KUKA KRL program: MyProgram_187().src

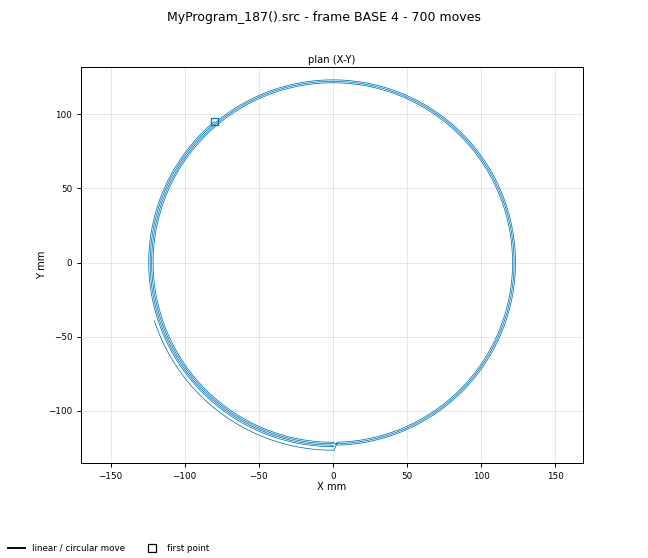
[picture p0: tool path of MyProgram_187().src in frame BASE 4, 700 of 700 moves have a stored position in this frame; points joined in program order, loops and branches not executed]
&ACCESS RVP
&REL 1
&PARAM TEMPLATE = C:\KRC\Roboter\Template\vorgabe
&PARAM EDITMASK = *
DEF MyProgram_187()
; ---- Setting reference (Base) ----
$BASE = BASE_DATA[4]

; --------------------------
; ---- Setting tool (TCP) ----
$TOOL = TOOL_DATA[3]
; --------------------------

$VEL.CP = VEL_APROX_PRINT
Startdeposition()
$VEL.CP = VEL_PRINT
LIN {X -79.8891,Y 95.1931,Z 136,A 126.8253,B 24.9437,C -1.7328,E1 24.8952,E2 319.3124} C_DIS
LIN {X -82.9171,Y 92.5676,Z 136,A 128.0656,B 24.9458,C -1.7009,E1 24.8928,E2 318.1432} C_DIS
LIN {X -85.2683,Y 90.4064,Z 136,A 130.1742,B 24.9442,C -1.7263,E1 24.8883,E2 315.9655} C_DIS
LIN {X -88.1797,Y 87.569,Z 136,A 131.451,B 24.9462,C -1.6946,E1 24.8859,E2 314.7588} C_DIS
LIN {X -91.7827,Y 83.7859,Z 136,A 133.7953,B 24.9468,C -1.6855,E1 24.8815,E2 312.4257} C_DIS
LIN {X -93.7322,Y 81.5983,Z 136,A 135.6415,B 24.9456,C -1.7044,E1 24.878,E2 310.5264} C_DIS
LIN {X -96.8546,Y 77.8667,Z 136,A 137.691,B 24.9465,C -1.6896,E1 24.8744,E2 308.5025} C_DIS
LIN {X -99.4155,Y 74.57,Z 136,A 139.5341,B 24.9471,C -1.6807,E1 24.8713,E2 306.6719} C_DIS
LIN {X -101.7751,Y 71.316,Z 136,A 141.5268,B 24.947,C -1.6818,E1 24.868,E2 304.6668} C_DIS
LIN {X -106.6362,Y 63.8183,Z 136,A 145.6095,B 24.9478,C -1.6682,E1 24.862,E2 300.5958} C_DIS
LIN {X -108.656,Y 60.3149,Z 136,A 148.5211,B 24.9452,C -1.71,E1 24.8579,E2 297.5692} C_DIS
LIN {X -111.8576,Y 54.1463,Z 136,A 150.5626,B 24.9491,C -1.6478,E1 24.8555,E2 295.6649} C_DIS
LIN {X -113.7433,Y 50.0655,Z 136,A 152.8918,B 24.9488,C -1.6529,E1 24.8528,E2 293.3109} C_DIS
LIN {X -115.0922,Y 46.8781,Z 136,A 154.451,B 24.9492,C -1.6463,E1 24.8511,E2 291.7587} C_DIS
LIN {X -116.506,Y 43.2441,Z 136,A 156.1505,B 24.9498,C -1.6363,E1 24.8494,E2 290.0735} C_DIS
LIN {X -117.7616,Y 39.6986,Z 136,A 157.9661,B 24.9499,C -1.6345,E1 24.8478,E2 288.252} C_DIS
LIN {X -119.6271,Y 33.6598,Z 136,A 160.8557,B 24.9506,C -1.624,E1 24.8455,E2 285.3706} C_DIS
LIN {X -120.6131,Y 29.9417,Z 136,A 162.772,B 24.9506,C -1.6246,E1 24.8441,E2 283.4416} C_DIS
LIN {X -122.2013,Y 22.6033,Z 136,A 166.0422,B 24.9517,C -1.6048,E1 24.8423,E2 280.1995} C_DIS
LIN {X -122.7677,Y 19.2815,Z 136,A 168.2135,B 24.9504,C -1.6274,E1 24.8413,E2 277.9615} C_DIS
LIN {X -123.363,Y 15.0101,Z 136,A 169.4402,B 24.9528,C -1.5868,E1 24.8409,E2 276.8241} C_DIS
LIN {X -123.9667,Y 8.7196,Z 136,A 172.4895,B 24.953,C -1.5832,E1 24.8402,E2 273.7651} C_DIS
LIN {X -124.135,Y 5.8576,Z 136,A 174.6101,B 24.9512,C -1.6146,E1 24.8399,E2 271.5569} C_DIS
LIN {X -124.2692,Y 0.9531,Z 136,A 176.6101,B 24.9523,C -1.5954,E1 24.8398,E2 269.5907} C_DIS
LIN {X -124.2442,Y -2.7393,Z 136,A 177.8627,B 24.9538,C -1.5697,E1 24.8398,E2 268.3918} C_DIS
LIN {X -124.1486,Y -5.5878,Z 136,A 179.9613,B 24.952,C -1.6006,E1 24.8402,E2 266.2069} C_DIS
LIN {X -123.821,Y -10.5841,Z 136,A -178.8273,B 24.9553,C -1.544,E1 24.8404,E2 265.1232} C_DIS
LIN {X -123.4086,Y -14.6276,Z 136,A -176.2872,B 24.954,C -1.5675,E1 24.8412,E2 262.5116} C_DIS
LIN {X -122.8522,Y -18.7364,Z 136,A -174.2614,B 24.954,C -1.5665,E1 24.842,E2 260.4763} C_DIS
LIN {X -122.3029,Y -22.0373,Z 136,A -172.7355,B 24.9544,C -1.5608,E1 24.8427,E2 258.9548} C_DIS
LIN {X -121.6747,Y -25.2814,Z 136,A -171.4403,B 24.9552,C -1.5458,E1 24.8434,E2 257.6879} C_DIS
LIN {X -120.8012,Y -29.1664,Z 136,A -169.6992,B 24.9558,C -1.5357,E1 24.8445,E2 255.9605} C_DIS
LIN {X -120.0039,Y -32.2916,Z 136,A -168.1059,B 24.9558,C -1.5359,E1 24.8457,E2 254.3576} C_DIS
LIN {X -118.874,Y -36.2296,Z 136,A -166.2328,B 24.9562,C -1.5293,E1 24.8472,E2 252.4893} C_DIS
LIN {X -117.8387,Y -39.4671,Z 136,A -164.6808,B 24.9565,C -1.5239,E1 24.8485,E2 250.9413} C_DIS
LIN {X -115.5921,Y -45.634,Z 136,A -161.576,B 24.9568,C -1.5183,E1 24.8516,E2 247.8323} C_DIS
LIN {X -114.1378,Y -49.1543,Z 136,A -159.2051,B 24.9555,C -1.5411,E1 24.8542,E2 245.3941} C_DIS
LIN {X -112.087,Y -53.6662,Z 136,A -157.5832,B 24.9576,C -1.5044,E1 24.8561,E2 243.8508} C_DIS
LIN {X -110.4867,Y -56.8906,Z 136,A -155.7892,B 24.9576,C -1.5058,E1 24.8584,E2 242.0439} C_DIS
LIN {X -107.6039,Y -62.1724,Z 136,A -153.0618,B 24.9581,C -1.496,E1 24.8621,E2 239.3255} C_DIS
LIN {X -105.3899,Y -65.8561,Z 136,A -150.667,B 24.9573,C -1.5095,E1 24.8656,E2 236.8863} C_DIS
LIN {X -103.2575,Y -69.1515,Z 136,A -149.3057,B 24.9587,C -1.4843,E1 24.8677,E2 235.5781} C_DIS
LIN {X -101.0566,Y -72.3296,Z 136,A -147.4329,B 24.9587,C -1.4839,E1 24.8707,E2 233.6972} C_DIS
LIN {X -97.1018,Y -77.5583,Z 136,A -144.667,B 24.9598,C -1.4647,E1 24.8753,E2 230.9637} C_DIS
LIN {X -95.265,Y -79.8034,Z 136,A -142.5722,B 24.9581,C -1.4963,E1 24.8792,E2 228.7842} C_DIS
LIN {X -92.3581,Y -83.151,Z 136,A -141.2515,B 24.9602,C -1.4582,E1 24.8815,E2 227.548} C_DIS
LIN {X -90.2674,Y -85.4156,Z 136,A -139.6102,B 24.9598,C -1.4652,E1 24.8847,E2 225.883} C_DIS
LIN {X -87.4192,Y -88.3286,Z 136,A -137.2447,B 24.9588,C -1.4836,E1 24.8895,E2 223.4636} C_DIS
LIN {X -84.3632,Y -91.2522,Z 136,A -135.706,B 24.96,C -1.4605,E1 24.8925,E2 221.9737} C_DIS
LIN {X -81.1483,Y -94.122,Z 136,A -133.2473,B 24.959,C -1.4785,E1 24.8978,E2 219.4625} C_DIS
LIN {X -77.7238,Y -96.9698,Z 136,A -131.922,B 24.9611,C -1.4407,E1 24.9005,E2 218.222} C_DIS
LIN {X -75.1964,Y -98.9426,Z 136,A -130.1587,B 24.9605,C -1.4513,E1 24.9045,E2 216.4273} C_DIS
LIN {X -71.5559,Y -101.6059,Z 136,A -128.1016,B 24.9608,C -1.4466,E1 24.9091,E2 214.374} C_DIS
LIN {X -68.0094,Y -104.0138,Z 136,A -126.0821,B 24.9608,C -1.4454,E1 24.9138,E2 212.3507} C_DIS
LIN {X -64.3396,Y -106.3222,Z 136,A -123.9135,B 24.9606,C -1.4504,E1 24.919,E2 210.1637} C_DIS
LIN {X -61.0887,Y -108.223,Z 136,A -122.3702,B 24.9612,C -1.4388,E1 24.9227,E2 208.6433} C_DIS
LIN {X -57.4568,Y -110.1925,Z 136,A -120.5659,B 24.9616,C -1.4315,E1 24.9271,E2 206.8512} C_DIS
LIN {X -54.7157,Y -111.5787,Z 136,A -119.0959,B 24.9616,C -1.4323,E1 24.9308,E2 205.3755} C_DIS
LIN {X -50.9574,Y -113.3444,Z 136,A -117.1344,B 24.9616,C -1.4323,E1 24.9358,E2 203.4092} C_DIS
LIN {X -47.7662,Y -114.7256,Z 136,A -115.5672,B 24.9618,C -1.4289,E1 24.9398,E2 201.8465} C_DIS
LIN {X -44.3758,Y -116.0812,Z 136,A -113.7716,B 24.9616,C -1.4325,E1 24.9445,E2 200.0384} C_DIS
LIN {X -40.7055,Y -117.4165,Z 136,A -112.0488,B 24.9618,C -1.4273,E1 24.9491,E2 198.3247} C_DIS
LIN {X -35.3019,Y -119.1534,Z 136,A -109.6672,B 24.9625,C -1.414,E1 24.9553,E2 195.9703} C_DIS
LIN {X -28.6712,Y -120.9205,Z 136,A -106.2014,B 24.9619,C -1.4265,E1 24.9648,E2 192.4698} C_DIS
LIN {X -24.5204,Y -121.8295,Z 136,A -104.3549,B 24.9622,C -1.4202,E1 24.9698,E2 190.636} C_DIS
LIN {X -20.6183,Y -122.5501,Z 136,A -102.4802,B 24.9622,C -1.4218,E1 24.975,E2 188.7557} C_DIS
LIN {X -16.3953,Y -123.1864,Z 136,A -100.6001,B 24.9624,C -1.417,E1 24.9801,E2 186.8853} C_DIS
LIN {X -13.0699,Y -123.5835,Z 136,A -98.9872,B 24.9622,C -1.4201,E1 24.9846,E2 185.2641} C_DIS
LIN {X -9.0853,Y -123.94,Z 136,A -97.1631,B 24.9622,C -1.4191,E1 24.9897,E2 183.4417} C_DIS
LIN {X -5.3221,Y -124.1595,Z 136,A -95.3481,B 24.9621,C -1.4229,E1 24.9948,E2 181.617} C_DIS
LIN {X -1.8056,Y -124.2598,Z 136,A -93.7695,B 24.9621,C -1.4211,E1 24.9992,E2 180.0426} C_DIS
LIN {X 0.8741,Y -124.2669,Z 136,A -92.7926,B 24.9628,C -1.4088,E1 25.0018,E2 179.0948} C_DIS
Enddeposition()
LIN {X 0.8741,Y -124.2669,Z 136,A -92.7926,B 24.9628,C -1.4088,E1 25.0018,E2 179.0948} C_DIS
Startdeposition()
$VEL.CP = VEL_PRINT
LIN {X -0.7971,Y -123.2805,Z 136,A -94.1303,B 24.9633,C -1.399,E1 24.998,E2 180.4558} C_DIS
LIN {X -4.8298,Y -123.1883,Z 136,A -95.9638,B 24.9633,C -1.4007,E1 24.9929,E2 182.2855} C_DIS
LIN {X -8.7858,Y -122.9696,Z 136,A -97.8638,B 24.9633,C -1.3979,E1 24.9876,E2 184.1928} C_DIS
LIN {X -13.0721,Y -122.5879,Z 136,A -99.8139,B 24.9633,C -1.4004,E1 24.9822,E2 186.1379} C_DIS
LIN {X -17.0591,Y -122.0974,Z 136,A -101.7751,B 24.9635,C -1.3964,E1 24.9767,E2 188.1103} C_DIS
LIN {X -20.0684,Y -121.6386,Z 136,A -103.1354,B 24.9633,C -1.3993,E1 24.973,E2 189.4648} C_DIS
LIN {X -23.7259,Y -120.9796,Z 136,A -104.9841,B 24.9636,C -1.3943,E1 24.9679,E2 191.3275} C_DIS
LIN {X -27.3955,Y -120.2003,Z 136,A -106.8949,B 24.9639,C -1.3874,E1 24.9626,E2 193.2571} C_DIS
LIN {X -30.6506,Y -119.4122,Z 136,A -108.2094,B 24.9633,C -1.3995,E1 24.9592,E2 194.5446} C_DIS
LIN {X -38.1177,Y -117.2435,Z 136,A -111.681,B 24.9628,C -1.4087,E1 24.9499,E2 198.0003} C_DIS
LIN {X -41.2854,Y -116.1655,Z 136,A -113.3984,B 24.9632,C -1.4025,E1 24.9453,E2 199.7358} C_DIS
LIN {X -44.7539,Y -114.8724,Z 136,A -115.0596,B 24.9629,C -1.4069,E1 24.941,E2 201.39} C_DIS
LIN {X -48.0441,Y -113.5371,Z 136,A -116.5953,B 24.9626,C -1.4139,E1 24.9371,E2 202.9126} C_DIS
LIN {X -50.4756,Y -112.4758,Z 136,A -117.9131,B 24.9626,C -1.4114,E1 24.9337,E2 204.2395} C_DIS
LIN {X -53.3978,Y -111.1185,Z 136,A -119.3608,B 24.9625,C -1.4154,E1 24.9301,E2 205.6812} C_DIS
LIN {X -56.2779,Y -109.6882,Z 136,A -120.8925,B 24.9625,C -1.4156,E1 24.9262,E2 207.2165} C_DIS
LIN {X -59.2874,Y -108.0931,Z 136,A -122.5495,B 24.9625,C -1.4144,E1 24.9221,E2 208.8812} C_DIS
LIN {X -62.877,Y -106.0443,Z 136,A -124.6374,B 24.9628,C -1.4095,E1 24.9171,E2 210.9869} C_DIS
LIN {X -66.1805,Y -104.0157,Z 136,A -126.3077,B 24.9623,C -1.4183,E1 24.9131,E2 212.6416} C_DIS
LIN {X -69.6137,Y -101.7496,Z 136,A -128.2574,B 24.9623,C -1.4197,E1 24.9086,E2 214.5944} C_DIS
LIN {X -73.3032,Y -99.1252,Z 136,A -130.3531,B 24.962,C -1.4237,E1 24.9039,E2 216.6879} C_DIS
LIN {X -76.6207,Y -96.5833,Z 136,A -132.9382,B 24.9634,C -1.3985,E1 24.8981,E2 219.3426} C_DIS
LIN {X -80.6051,Y -93.2838,Z 136,A -134.6338,B 24.9614,C -1.4349,E1 24.8946,E2 220.9581} C_DIS
LIN {X -83.5872,Y -90.6214,Z 136,A -137.0973,B 24.9627,C -1.4116,E1 24.8894,E2 223.487} C_DIS
LIN {X -86.899,Y -87.4504,Z 136,A -138.5028,B 24.9607,C -1.4486,E1 24.8868,E2 224.8104} C_DIS
LIN {X -89.289,Y -85.0091,Z 136,A -140.3163,B 24.9611,C -1.4419,E1 24.8832,E2 226.6476} C_DIS
LIN {X -94.242,Y -79.483,Z 136,A -143.5737,B 24.9602,C -1.4584,E1 24.8772,E2 229.8803} C_DIS
LIN {X -98.2148,Y -74.5182,Z 136,A -146.4389,B 24.9595,C -1.4696,E1 24.8723,E2 232.7324} C_DIS
LIN {X -99.7531,Y -72.4455,Z 136,A -147.9432,B 24.9601,C -1.459,E1 24.8697,E2 234.2692} C_DIS
LIN {X -102.2995,Y -68.8039,Z 136,A -150.822,B 24.9618,C -1.4286,E1 24.8651,E2 237.2347} C_DIS
LIN {X -105.4462,Y -63.8758,Z 136,A -153.3873,B 24.961,C -1.4425,E1 24.8614,E2 239.78} C_DIS
LIN {X -107.9909,Y -59.4732,Z 136,A -154.8402,B 24.9585,C -1.489,E1 24.8596,E2 241.1298} C_DIS
LIN {X -109.8808,Y -55.8996,Z 136,A -156.9074,B 24.9586,C -1.486,E1 24.8569,E2 243.2152} C_DIS
LIN {X -111.277,Y -53.0659,Z 136,A -159.3366,B 24.9607,C -1.4482,E1 24.8539,E2 245.7475} C_DIS
LIN {X -113.7429,Y -47.5514,Z 136,A -161.0675,B 24.9577,C -1.5034,E1 24.8521,E2 247.3566} C_DIS
LIN {X -116.1405,Y -41.3547,Z 136,A -164.2218,B 24.9573,C -1.5096,E1 24.8489,E2 250.5139} C_DIS
LIN {X -116.9716,Y -38.9387,Z 136,A -165.5697,B 24.9575,C -1.5062,E1 24.8477,E2 251.8776} C_DIS
LIN {X -118.0764,Y -35.4541,Z 136,A -167.3797,B 24.9575,C -1.5065,E1 24.8462,E2 253.6972} C_DIS
LIN {X -119.1135,Y -31.7896,Z 136,A -169.0301,B 24.9569,C -1.5172,E1 24.845,E2 255.3316} C_DIS
LIN {X -120.0435,Y -28.082,Z 136,A -170.9327,B 24.9569,C -1.5172,E1 24.8437,E2 257.2453} C_DIS
LIN {X -121.5095,Y -20.842,Z 136,A -174.1659,B 24.9557,C -1.5369,E1 24.842,E2 260.4509} C_DIS
LIN {X -122.1588,Y -16.6207,Z 136,A -176.9281,B 24.9573,C -1.5096,E1 24.8409,E2 263.2947} C_DIS
LIN {X -122.6999,Y -11.9764,Z 136,A -178.1992,B 24.9547,C -1.5557,E1 24.8406,E2 264.4634} C_DIS
LIN {X -123.0439,Y -7.6728,Z 136,A 179.2812,B 24.9556,C -1.5399,E1 24.84,E2 267.0358} C_DIS
LIN {X -123.2096,Y -4.2848,Z 136,A 177.075,B 24.9568,C -1.5179,E1 24.8398,E2 269.3077} C_DIS
LIN {X -123.2763,Y 1.43,Z 136,A 175.325,B 24.9541,C -1.5656,E1 24.8398,E2 270.9546} C_DIS
LIN {X -123.1001,Y 6.7344,Z 136,A 172.8345,B 24.9537,C -1.5726,E1 24.8401,E2 273.4433} C_DIS
LIN {X -122.5522,Y 13.4038,Z 136,A 169.7573,B 24.953,C -1.5842,E1 24.8408,E2 276.5113} C_DIS
LIN {X -121.7875,Y 19.1446,Z 136,A 166.9893,B 24.9526,C -1.5897,E1 24.8419,E2 279.2827} C_DIS
LIN {X -121.2402,Y 22.3575,Z 136,A 164.5557,B 24.9547,C -1.5551,E1 24.8432,E2 281.8134} C_DIS
LIN {X -120.0973,Y 27.8462,Z 136,A 162.8245,B 24.952,C -1.6011,E1 24.8442,E2 283.445} C_DIS
LIN {X -119.3463,Y 30.9102,Z 136,A 161.235,B 24.952,C -1.6005,E1 24.8452,E2 285.0453} C_DIS
LIN {X -118.0768,Y 35.447,Z 136,A 158.561,B 24.9528,C -1.5866,E1 24.8474,E2 287.7678} C_DIS
LIN {X -116.784,Y 39.5023,Z 136,A 157.1951,B 24.9509,C -1.6193,E1 24.8485,E2 289.0635} C_DIS
LIN {X -115.2983,Y 43.6472,Z 136,A 155.0459,B 24.9507,C -1.6213,E1 24.8506,E2 291.2201} C_DIS
LIN {X -113.8043,Y 47.4042,Z 136,A 153.1553,B 24.9504,C -1.6267,E1 24.8526,E2 293.1085} C_DIS
LIN {X -112.4721,Y 50.4839,Z 136,A 151.5761,B 24.9502,C -1.6306,E1 24.8543,E2 294.687} C_DIS
LIN {X -111.1031,Y 53.43,Z 136,A 149.5201,B 24.9513,C -1.6115,E1 24.8569,E2 296.7995} C_DIS
LIN {X -109.2176,Y 57.1847,Z 136,A 147.6227,B 24.9508,C -1.6198,E1 24.8593,E2 298.6874} C_DIS
LIN {X -107.2843,Y 60.7392,Z 136,A 146.388,B 24.9488,C -1.6534,E1 24.8609,E2 299.8486} C_DIS
LIN {X -102.6336,Y 68.3036,Z 136,A 142.0902,B 24.9485,C -1.6578,E1 24.8673,E2 304.1578} C_DIS
LIN {X -100.536,Y 71.3559,Z 136,A 140.2133,B 24.9486,C -1.6558,E1 24.8703,E2 306.0487} C_DIS
LIN {X -97.7397,Y 75.1402,Z 136,A 138.1224,B 24.948,C -1.666,E1 24.8737,E2 308.1254} C_DIS
LIN {X -95.4028,Y 78.0854,Z 136,A 136.0344,B 24.9486,C -1.6558,E1 24.8775,E2 310.2475} C_DIS
LIN {X -93.3376,Y 80.5426,Z 136,A 135.0727,B 24.9469,C -1.6829,E1 24.8791,E2 311.1489} C_DIS
LIN {X -91.5279,Y 82.594,Z 136,A 133.137,B 24.9485,C -1.657,E1 24.8828,E2 313.1549} C_DIS
LIN {X -88.9686,Y 85.3443,Z 136,A 131.8356,B 24.9471,C -1.6809,E1 24.8853,E2 314.4052} C_DIS
LIN {X -85.0552,Y 89.2449,Z 136,A 129.4074,B 24.9463,C -1.6933,E1 24.89,E2 316.8139} C_DIS
LIN {X -82.7792,Y 91.3598,Z 136,A 127.5149,B 24.9473,C -1.6769,E1 24.894,E2 318.7531} C_DIS
LIN {X -80.0922,Y 93.7249,Z 136,A 126.0172,B 24.9466,C -1.688,E1 24.8972,E2 320.2302} C_DIS
LIN {X -75.2732,Y 97.6374,Z 136,A 123.1518,B 24.9461,C -1.6952,E1 24.9034,E2 323.0892} C_DIS
LIN {X -71.9619,Y 100.1029,Z 136,A 120.9433,B 24.9467,C -1.6864,E1 24.9084,E2 325.3265} C_DIS
LIN {X -69.2441,Y 102.0014,Z 136,A 119.1971,B 24.9471,C -1.6804,E1 24.9125,E2 327.0927} C_DIS
LIN {X -65.6679,Y 104.3395,Z 136,A 117.7502,B 24.9453,C -1.7081,E1 24.9158,E2 328.4783} C_DIS
LIN {X -62.2817,Y 106.3957,Z 136,A 115.7431,B 24.9456,C -1.7041,E1 24.9206,E2 330.501} C_DIS
LIN {X -58.7148,Y 108.4053,Z 136,A 113.8957,B 24.9452,C -1.7099,E1 24.9251,E2 332.34} C_DIS
LIN {X -55.6171,Y 110.0246,Z 136,A 112.3365,B 24.9448,C -1.7156,E1 24.929,E2 333.8899} C_DIS
LIN {X -51.8752,Y 111.8372,Z 136,A 110.3993,B 24.9447,C -1.7185,E1 24.9339,E2 335.8252} C_DIS
LIN {X -46.0929,Y 114.3417,Z 136,A 107.836,B 24.9433,C -1.7393,E1 24.9404,E2 338.3451} C_DIS
LIN {X -42.9145,Y 115.5727,Z 136,A 105.8955,B 24.9442,C -1.7252,E1 24.9455,E2 340.323} C_DIS
LIN {X -38.5445,Y 117.1029,Z 136,A 103.7789,B 24.9439,C -1.7295,E1 24.9511,E2 342.4335} C_DIS
LIN {X -35.6805,Y 118.0071,Z 136,A 102.3388,B 24.9439,C -1.7291,E1 24.9549,E2 343.8771} C_DIS
LIN {X -29.2711,Y 119.758,Z 136,A 99.4324,B 24.9432,C -1.7406,E1 24.9627,E2 346.7607} C_DIS
LIN {X -27.0063,Y 120.2889,Z 136,A 97.6434,B 24.9452,C -1.7093,E1 24.9678,E2 348.6262} C_DIS
LIN {X -22.9703,Y 121.124,Z 136,A 96.5296,B 24.9428,C -1.7475,E1 24.9706,E2 349.6506} C_DIS
LIN {X -20.395,Y 121.5841,Z 136,A 94.3114,B 24.9457,C -1.7026,E1 24.977,E2 351.9775} C_DIS
LIN {X -15.2822,Y 122.3339,Z 136,A 92.6842,B 24.9433,C -1.7394,E1 24.9813,E2 353.5186} C_DIS
LIN {X -10.9994,Y 122.7928,Z 136,A 90.4986,B 24.9438,C -1.732,E1 24.9874,E2 355.723} C_DIS
LIN {X -7.0479,Y 123.0824,Z 136,A 88.6722,B 24.9437,C -1.7334,E1 24.9925,E2 357.5466} C_DIS
LIN {X -3.1815,Y 123.2421,Z 136,A 86.9936,B 24.9433,C -1.7395,E1 24.9971,E2 359.2109} C_DIS
LIN {X 0.5109,Y 123.2821,Z 136,A 85.2323,B 24.9434,C -1.7378,E1 25.002,E2 360.9764} C_DIS
LIN {X 4.5588,Y 123.1989,Z 136,A 83.3503,B 24.9434,C -1.738,E1 25.0073,E2 362.8575} C_DIS
LIN {X 8.0968,Y 123.0178,Z 136,A 81.6549,B 24.9435,C -1.7357,E1 25.012,E2 364.5577} C_DIS
LIN {X 11.8511,Y 122.7119,Z 136,A 79.9012,B 24.9435,C -1.7354,E1 25.0169,E2 366.3111} C_DIS
LIN {X 16.386,Y 122.1895,Z 136,A 77.8547,B 24.9434,C -1.7385,E1 25.0225,E2 368.3487} C_DIS
LIN {X 20.1788,Y 121.6202,Z 136,A 75.7807,B 24.9443,C -1.7242,E1 25.0284,E2 370.4544} C_DIS
LIN {X 23.9354,Y 120.9387,Z 136,A 74.2502,B 24.9436,C -1.7349,E1 25.0325,E2 371.9578} C_DIS
LIN {X 26.8973,Y 120.3141,Z 136,A 73.0086,B 24.9431,C -1.742,E1 25.0358,E2 373.181} C_DIS
LIN {X 29.837,Y 119.6187,Z 136,A 70.7055,B 24.9459,C -1.6988,E1 25.0423,E2 375.5829} C_DIS
LIN {X 35.0837,Y 118.1861,Z 136,A 69.1007,B 24.9432,C -1.7406,E1 25.0464,E2 377.0863} C_DIS
LIN {X 37.5544,Y 117.4234,Z 136,A 67.7868,B 24.9436,C -1.7343,E1 25.0499,E2 378.4126} C_DIS
LIN {X 41.1043,Y 116.2308,Z 136,A 65.8924,B 24.9442,C -1.7254,E1 25.0549,E2 380.3243} C_DIS
LIN {X 44.6198,Y 114.9246,Z 136,A 64.3147,B 24.9438,C -1.7316,E1 25.059,E2 381.884} C_DIS
LIN {X 47.8018,Y 113.6383,Z 136,A 62.7298,B 24.9438,C -1.7304,E1 25.0631,E2 383.468} C_DIS
LIN {X 51.0017,Y 112.2405,Z 136,A 60.8741,B 24.9447,C -1.7173,E1 25.0679,E2 385.3501} C_DIS
LIN {X 54.6188,Y 110.5231,Z 136,A 59.218,B 24.9442,C -1.7248,E1 25.072,E2 386.984} C_DIS
LIN {X 57.6727,Y 108.9613,Z 136,A 57.6108,B 24.9444,C -1.7221,E1 25.076,E2 388.5933} C_DIS
LIN {X 61.2582,Y 106.9883,Z 136,A 55.5187,B 24.9452,C -1.7101,E1 25.0811,E2 390.7074} C_DIS
LIN {X 64.532,Y 105.0459,Z 136,A 53.9147,B 24.9449,C -1.7154,E1 25.0849,E2 392.2939} C_DIS
LIN {X 67.9392,Y 102.8752,Z 136,A 52.0488,B 24.945,C -1.7129,E1 25.0893,E2 394.1596} C_DIS
LIN {X 71.3905,Y 100.5114,Z 136,A 50.0353,B 24.9454,C -1.7062,E1 25.0939,E2 396.1819} C_DIS
LIN {X 75.2954,Y 97.6192,Z 136,A 47.5381,B 24.9464,C -1.6906,E1 25.0995,E2 398.7071} C_DIS
LIN {X 78.0673,Y 95.4176,Z 136,A 46.4356,B 24.945,C -1.7139,E1 25.1018,E2 399.7504} C_DIS
LIN {X 80.3223,Y 93.5274,Z 136,A 44.8089,B 24.9459,C -1.6985,E1 25.1053,E2 401.4072} C_DIS
LIN {X 83.5894,Y 90.6194,Z 136,A 42.8267,B 24.946,C -1.6968,E1 25.1094,E2 403.3854} C_DIS
LIN {X 86.6269,Y 87.7208,Z 136,A 40.8362,B 24.9464,C -1.6907,E1 25.1134,E2 405.382} C_DIS
LIN {X 89.9028,Y 84.3589,Z 136,A 38.4815,B 24.9473,C -1.6773,E1 25.118,E2 407.7581} C_DIS
LIN {X 92.5137,Y 81.4879,Z 136,A 36.8883,B 24.9469,C -1.6835,E1 25.1209,E2 409.3296} C_DIS
LIN {X 95.2199,Y 78.309,Z 136,A 34.9921,B 24.947,C -1.681,E1 25.1243,E2 411.223} C_DIS
LIN {X 97.7627,Y 75.1102,Z 136,A 33.0687,B 24.9474,C -1.6751,E1 25.1276,E2 413.1511} C_DIS
LIN {X 100.2457,Y 71.7622,Z 136,A 31.1524,B 24.9477,C -1.6713,E1 25.1308,E2 415.0673} C_DIS
LIN {X 102.7626,Y 68.1103,Z 136,A 29.0612,B 24.9481,C -1.6644,E1 25.1341,E2 417.1643} C_DIS
LIN {X 105.1582,Y 64.349,Z 136,A 27.0529,B 24.9482,C -1.6621,E1 25.137,E2 419.168} C_DIS
LIN {X 107.309,Y 60.6951,Z 136,A 25.0597,B 24.9486,C -1.6555,E1 25.1398,E2 421.1663} C_DIS
LIN {X 109.3355,Y 56.9601,Z 136,A 23.2234,B 24.9486,C -1.657,E1 25.1422,E2 422.9896} C_DIS
LIN {X 110.9331,Y 53.7859,Z 136,A 21.0139,B 24.9506,C -1.6244,E1 25.145,E2 425.264} C_DIS
LIN {X 112.7251,Y 49.9181,Z 136,A 19.6538,B 24.949,C -1.6496,E1 25.1465,E2 426.5573} C_DIS
LIN {X 113.8281,Y 47.3473,Z 136,A 18.286,B 24.9495,C -1.6424,E1 25.148,E2 427.9345} C_DIS
LIN {X 115.3108,Y 43.6138,Z 136,A 16.4069,B 24.9498,C -1.6362,E1 25.1499,E2 429.8178} C_DIS
LIN {X 116.4617,Y 40.4383,Z 136,A 14.9034,B 24.9499,C -1.6348,E1 25.1513,E2 431.3161} C_DIS
LIN {X 118.8182,Y 32.8778,Z 136,A 11.1306,B 24.9509,C -1.6188,E1 25.1544,E2 435.1052} C_DIS
LIN {X 120.2244,Y 27.2899,Z 136,A 8.4179,B 24.9515,C -1.6086,E1 25.1562,E2 437.8262} C_DIS
LIN {X 121.6217,Y 20.1694,Z 136,A 5.2082,B 24.9517,C -1.6061,E1 25.1578,E2 441.0232} C_DIS
LIN {X 122.2843,Y 15.6626,Z 136,A 3.2015,B 24.9517,C -1.6048,E1 25.1586,E2 443.021} C_DIS
LIN {X 122.5732,Y 13.209,Z 136,A 1.9814,B 24.9522,C -1.5975,E1 25.159,E2 444.2512} C_DIS
LIN {X 122.9105,Y 9.5956,Z 136,A 0.1999,B 24.9528,C -1.5872,E1 25.1594,E2 446.0464} C_DIS
LIN {X 123.1431,Y 5.8773,Z 136,A -1.4797,B 24.953,C -1.5842,E1 25.1597,E2 447.7231} C_DIS
LIN {X 123.268,Y 1.9235,Z 136,A -3.2531,B 24.9531,C -1.5814,E1 25.1597,E2 449.4925} C_DIS
LIN {X 123.2658,Y -2.0555,Z 136,A -5.0751,B 24.9534,C -1.5767,E1 25.1597,E2 451.3146} C_DIS
LIN {X 123.1436,Y -5.8679,Z 136,A -6.9014,B 24.9539,C -1.5682,E1 25.1595,E2 453.1502} C_DIS
LIN {X 122.8768,Y -10.0051,Z 136,A -8.8377,B 24.9543,C -1.5614,E1 25.1592,E2 455.0911} C_DIS
LIN {X 122.4882,Y -13.9882,Z 136,A -10.6975,B 24.9547,C -1.5552,E1 25.1586,E2 456.9544} C_DIS
LIN {X 122.002,Y -17.7267,Z 136,A -12.4439,B 24.955,C -1.5498,E1 25.1579,E2 458.7034} C_DIS
LIN {X 121.3479,Y -21.7557,Z 136,A -14.2306,B 24.955,C -1.5492,E1 25.1571,E2 460.481} C_DIS
LIN {X 120.4026,Y -26.4967,Z 136,A -16.5301,B 24.9556,C -1.5391,E1 25.1558,E2 462.7907} C_DIS
LIN {X 119.5011,Y -30.3002,Z 136,A -18.267,B 24.9557,C -1.5373,E1 25.1546,E2 464.5219} C_DIS
LIN {X 118.5106,Y -33.9753,Z 136,A -20.9295,B 24.9586,C -1.4867,E1 25.1525,E2 467.2885} C_DIS
LIN {X 116.6947,Y -39.7662,Z 136,A -22.7395,B 24.9562,C -1.5284,E1 25.151,E2 468.9899} C_DIS
LIN {X 115.365,Y -43.4691,Z 136,A -24.6424,B 24.9568,C -1.5189,E1 25.1492,E2 470.9045} C_DIS
LIN {X 112.7492,Y -49.8642,Z 136,A -27.6899,B 24.9568,C -1.5171,E1 25.146,E2 473.9394} C_DIS
LIN {X 111.2087,Y -53.209,Z 136,A -29.4819,B 24.9574,C -1.5078,E1 25.1438,E2 475.7437} C_DIS
LIN {X 108.7471,Y -58.0782,Z 136,A -32.0419,B 24.9579,C -1.4989,E1 25.1406,E2 478.3112} C_DIS
LIN {X 107.4753,Y -60.3992,Z 136,A -33.3556,B 24.9584,C -1.491,E1 25.1387,E2 479.6367} C_DIS
LIN {X 105.2688,Y -64.1687,Z 136,A -35.7157,B 24.9596,C -1.4684,E1 25.1353,E2 482.0378} C_DIS
LIN {X 103.2715,Y -67.3356,Z 136,A -36.8724,B 24.9583,C -1.4927,E1 25.1336,E2 483.1314} C_DIS
LIN {X 100.3985,Y -71.5485,Z 136,A -39.3319,B 24.9589,C -1.4815,E1 25.1297,E2 485.6054} C_DIS
LIN {X 98.2955,Y -74.4107,Z 136,A -41.142,B 24.9596,C -1.4689,E1 25.1267,E2 487.4365} C_DIS
LIN {X 95.965,Y -77.3933,Z 136,A -43.0619,B 24.9603,C -1.4561,E1 25.1233,E2 489.3777} C_DIS
LIN {X 92.4118,Y -81.6032,Z 136,A -45.39,B 24.96,C -1.4609,E1 25.1191,E2 491.6838} C_DIS
LIN {X 89.487,Y -84.8007,Z 136,A -47.6304,B 24.9609,C -1.4445,E1 25.1147,E2 493.9532} C_DIS
LIN {X 87.2261,Y -87.1247,Z 136,A -49.0699,B 24.9609,C -1.4441,E1 25.1119,E2 495.3875} C_DIS
LIN {X 84.2892,Y -89.9694,Z 136,A -50.7809,B 24.9607,C -1.4489,E1 25.1085,E2 497.0801} C_DIS
LIN {X 80.1903,Y -93.6402,Z 136,A -53.4138,B 24.9612,C -1.4391,E1 25.1029,E2 499.7256} C_DIS
LIN {X 76.4504,Y -96.7186,Z 136,A -55.6152,B 24.9613,C -1.4366,E1 25.0982,E2 501.9248} C_DIS
LIN {X 72.9054,Y -99.4175,Z 136,A -58.3817,B 24.9634,C -1.3979,E1 25.0918,E2 504.7728} C_DIS
LIN {X 68.2172,Y -102.6913,Z 136,A -60.8335,B 24.9632,C -1.4026,E1 25.0861,E2 507.2054} C_DIS
LIN {X 64.1861,Y -105.2581,Z 136,A -62.1583,B 24.961,C -1.4424,E1 25.0832,E2 508.4318} C_DIS
LIN {X 60.242,Y -107.5637,Z 136,A -64.9452,B 24.963,C -1.4058,E1 25.0763,E2 511.2969} C_DIS
LIN {X 57.0538,Y -109.2863,Z 136,A -66.7555,B 24.9635,C -1.3968,E1 25.0717,E2 513.1234} C_DIS
LIN {X 53.1586,Y -111.2327,Z 136,A -68.1935,B 24.9621,C -1.4221,E1 25.0683,E2 514.4978} C_DIS
LIN {X 45.6218,Y -114.5316,Z 136,A -71.9656,B 24.9623,C -1.4188,E1 25.0586,E2 518.2687} C_DIS
LIN {X 43.1448,Y -115.4864,Z 136,A -73.2396,B 24.9625,C -1.4151,E1 25.0553,E2 519.5486} C_DIS
LIN {X 39.6073,Y -116.749,Z 136,A -76.0752,B 24.9653,C -1.3602,E1 25.0475,E2 522.5085} C_DIS
LIN {X 33.114,Y -118.7522,Z 136,A -78.0897,B 24.9627,C -1.4117,E1 25.0424,E2 524.3978} C_DIS
LIN {X 30.011,Y -119.5745,Z 136,A -80.1416,B 24.9642,C -1.3831,E1 25.0367,E2 526.5143} C_DIS
LIN {X 26.0247,Y -120.5045,Z 136,A -82.0179,B 24.9642,C -1.3826,E1 25.0315,E2 528.3893} C_DIS
LIN {X 22.0606,Y -121.2934,Z 136,A -83.2019,B 24.9625,C -1.4144,E1 25.0285,E2 529.4966} C_DIS
LIN {X 17.983,Y -121.9654,Z 136,A -85.3782,B 24.9633,C -1.4006,E1 25.0224,E2 531.7035} C_DIS
LIN {X 14.3981,Y -122.4393,Z 136,A -87.0795,B 24.9633,C -1.3986,E1 25.0177,E2 533.4083} C_DIS
LIN {X 10.4934,Y -122.8355,Z 136,A -88.8415,B 24.9633,C -1.4006,E1 25.0128,E2 535.1645} C_DIS
LIN {X 7.2186,Y -123.0719,Z 136,A -90.4395,B 24.9635,C -1.3965,E1 25.0083,E2 536.7715} C_DIS
LIN {X 3.2582,Y -123.24,Z 136,A -92.2671,B 24.9635,C -1.3965,E1 25.0032,E2 538.5986} C_DIS
LIN {X 3.2582,Y -123.24,Z 136,A -92.2671,B 24.9635,C -1.3965,E1 25.0032,E2 538.5986} C_DIS
Enddeposition()
LIN {X 0.8719,Y -122.2892,Z 136,A -93.284,B 24.9623,C -1.4181,E1 25.0005,E2 539.5643} C_DIS
Startdeposition()
$VEL.CP = VEL_PRINT
LIN {X 4.9775,Y -122.1922,Z 136,A -90.6693,B 24.9605,C -1.4516,E1 25.0081,E2 536.8707} C_DIS
LIN {X 8.8136,Y -121.9753,Z 136,A -88.8584,B 24.9605,C -1.4529,E1 25.0131,E2 535.0575} C_DIS
LIN {X 12.8168,Y -121.62,Z 136,A -86.953,B 24.9603,C -1.455,E1 25.0184,E2 533.1483} C_DIS
LIN {X 17.0537,Y -121.0985,Z 136,A -84.9998,B 24.9603,C -1.4541,E1 25.0238,E2 531.1989} C_DIS
LIN {X 20.7767,Y -120.5171,Z 136,A -83.3181,B 24.9605,C -1.4513,E1 25.0284,E2 529.5254} C_DIS
LIN {X 24.1435,Y -119.8864,Z 136,A -81.5449,B 24.96,C -1.4609,E1 25.0333,E2 527.7315} C_DIS
LIN {X 28.5926,Y -118.9036,Z 136,A -79.5211,B 24.9602,C -1.4576,E1 25.0388,E2 525.7185} C_DIS
LIN {X 32.0504,Y -118.0198,Z 136,A -77.7496,B 24.9598,C -1.4642,E1 25.0436,E2 523.9341} C_DIS
LIN {X 36.1049,Y -116.8423,Z 136,A -75.4997,B 24.959,C -1.4799,E1 25.0497,E2 521.6512} C_DIS
LIN {X 39.5336,Y -115.728,Z 136,A -74.131,B 24.9597,C -1.4662,E1 25.0533,E2 520.3173} C_DIS
LIN {X 42.9096,Y -114.5178,Z 136,A -72.5915,B 24.96,C -1.4616,E1 25.0573,E2 518.792} C_DIS
LIN {X 46.4141,Y -113.1452,Z 136,A -70.3755,B 24.9586,C -1.4864,E1 25.0631,E2 516.5223} C_DIS
LIN {X 49.5942,Y -111.7859,Z 136,A -69.1092,B 24.9594,C -1.4714,E1 25.0663,E2 515.2946} C_DIS
LIN {X 52.5031,Y -110.4492,Z 136,A -67.6604,B 24.9594,C -1.4714,E1 25.0699,E2 513.8497} C_DIS
LIN {X 55.296,Y -109.0776,Z 136,A -66.2834,B 24.9595,C -1.4698,E1 25.0733,E2 512.4801} C_DIS
LIN {X 60.3781,Y -106.351,Z 136,A -63.4126,B 24.9588,C -1.4829,E1 25.0804,E2 509.5867} C_DIS
LIN {X 63.9099,Y -104.2666,Z 136,A -61.374,B 24.9583,C -1.4924,E1 25.0853,E2 507.532} C_DIS
LIN {X 68.0469,Y -101.6151,Z 136,A -59.2113,B 24.9584,C -1.49,E1 25.0904,E2 505.3821} C_DIS
LIN {X 72.4362,Y -98.5342,Z 136,A -56.7343,B 24.9582,C -1.4935,E1 25.096,E2 502.9054} C_DIS
LIN {X 75.7369,Y -96.0207,Z 136,A -54.9435,B 24.9584,C -1.4901,E1 25.0999,E2 501.1292} C_DIS
LIN {X 78.3757,Y -93.8789,Z 136,A -52.6787,B 24.9563,C -1.5275,E1 25.1049,E2 498.7847} C_DIS
LIN {X 81.8848,Y -90.8351,Z 136,A -51.0323,B 24.9575,C -1.5059,E1 25.1083,E2 497.1959} C_DIS
LIN {X 84.884,Y -88.0384,Z 136,A -49.0987,B 24.9572,C -1.5112,E1 25.1122,E2 495.2578} C_DIS
LIN {X 88.0703,Y -84.851,Z 136,A -47.0279,B 24.957,C -1.5144,E1 25.1162,E2 493.1882} C_DIS
LIN {X 90.8819,Y -81.8325,Z 136,A -45.0659,B 24.9567,C -1.5209,E1 25.1199,E2 491.2197} C_DIS
LIN {X 93.522,Y -78.8016,Z 136,A -43.2143,B 24.9565,C -1.5243,E1 25.1233,E2 489.3685} C_DIS
LIN {X 95.8312,Y -75.9765,Z 136,A -41.1371,B 24.9551,C -1.5476,E1 25.127,E2 487.2461} C_DIS
LIN {X 98.2633,Y -72.8038,Z 136,A -39.701,B 24.9561,C -1.5306,E1 25.1293,E2 485.857} C_DIS
LIN {X 99.9625,Y -70.452,Z 136,A -38.2551,B 24.9556,C -1.5388,E1 25.1317,E2 484.3987} C_DIS
LIN {X 102.4791,Y -66.7387,Z 136,A -36.2252,B 24.9556,C -1.5412,E1 25.1348,E2 482.3734} C_DIS
LIN {X 104.9318,Y -62.812,Z 136,A -34.0658,B 24.9552,C -1.547,E1 25.1379,E2 480.2112} C_DIS
LIN {X 106.7464,Y -59.6764,Z 136,A -32.1027,B 24.9541,C -1.5656,E1 25.1407,E2 478.2144} C_DIS
LIN {X 108.3175,Y -56.7702,Z 136,A -30.9331,B 24.9549,C -1.551,E1 25.1421,E2 477.0854} C_DIS
LIN {X 109.9684,Y -53.5063,Z 136,A -29.2615,B 24.9548,C -1.554,E1 25.1442,E2 475.4156} C_DIS
LIN {X 111.4612,Y -50.3203,Z 136,A -27.5266,B 24.9542,C -1.5635,E1 25.1463,E2 473.6676} C_DIS
LIN {X 112.9516,Y -46.8781,Z 136,A -25.5663,B 24.9533,C -1.5793,E1 25.1484,E2 471.6809} C_DIS
LIN {X 114.8319,Y -42.0664,Z 136,A -23.3478,B 24.9534,C -1.5767,E1 25.1506,E2 469.481} C_DIS
LIN {X 116.0337,Y -38.6233,Z 136,A -21.4065,B 24.9524,C -1.594,E1 25.1523,E2 467.5098} C_DIS
LIN {X 117.0544,Y -35.4119,Z 136,A -20.0675,B 24.9528,C -1.5868,E1 25.1534,E2 466.1955} C_DIS
LIN {X 118.0661,Y -31.8768,Z 136,A -18.4651,B 24.9528,C -1.5862,E1 25.1546,E2 464.6035} C_DIS
LIN {X 118.8343,Y -28.88,Z 136,A -16.9694,B 24.9524,C -1.5933,E1 25.1556,E2 463.0999} C_DIS
LIN {X 119.7623,Y -24.7537,Z 136,A -15.257,B 24.9529,C -1.586,E1 25.1566,E2 461.4145} C_DIS
LIN {X 120.3764,Y -21.5671,Z 136,A -13.5391,B 24.952,C -1.601,E1 25.1575,E2 459.6713} C_DIS
LIN {X 120.8966,Y -18.431,Z 136,A -12.0712,B 24.9517,C -1.6048,E1 25.1581,E2 458.2031} C_DIS
LIN {X 121.4088,Y -14.6821,Z 136,A -10.2868,B 24.9514,C -1.6112,E1 25.1588,E2 456.4141} C_DIS
LIN {X 121.8134,Y -10.8367,Z 136,A -8.4373,B 24.9509,C -1.6191,E1 25.1593,E2 454.557} C_DIS
LIN {X 122.1019,Y -6.8698,Z 136,A -6.5522,B 24.9504,C -1.6263,E1 25.1596,E2 452.6661} C_DIS
LIN {X 122.2556,Y -3.0574,Z 136,A -4.8686,B 24.9504,C -1.6269,E1 25.1598,E2 450.9911} C_DIS
LIN {X 122.2941,Y 0.1575,Z 136,A -3.3587,B 24.9501,C -1.6321,E1 25.1598,E2 449.4781} C_DIS
LIN {X 122.2367,Y 3.7374,Z 136,A -1.6279,B 24.9496,C -1.6403,E1 25.1597,E2 447.7382} C_DIS
LIN {X 122.0481,Y 7.7441,Z 136,A 0.2394,B 24.9492,C -1.6458,E1 25.1594,E2 445.8689} C_DIS
LIN {X 121.7206,Y 11.8214,Z 136,A 2.0718,B 24.9492,C -1.6478,E1 25.1589,E2 444.0427} C_DIS
LIN {X 121.412,Y 14.6559,Z 136,A 3.807,B 24.9476,C -1.6725,E1 25.1583,E2 442.2597} C_DIS
LIN {X 120.9001,Y 18.4084,Z 136,A 4.9092,B 24.9494,C -1.644,E1 25.1579,E2 441.2311} C_DIS
LIN {X 120.5079,Y 20.83,Z 136,A 6.732,B 24.947,C -1.6818,E1 25.157,E2 439.3298} C_DIS
LIN {X 119.8092,Y 24.5228,Z 136,A 8.0435,B 24.9481,C -1.6646,E1 25.1563,E2 438.0666} C_DIS
LIN {X 118.6039,Y 29.8124,Z 136,A 10.5851,B 24.9476,C -1.6726,E1 25.1547,E2 435.5209} C_DIS
LIN {X 117.6952,Y 33.2192,Z 136,A 12.2077,B 24.9473,C -1.6762,E1 25.1535,E2 433.899} C_DIS
LIN {X 116.1078,Y 38.4006,Z 136,A 14.6875,B 24.947,C -1.681,E1 25.1514,E2 431.422} C_DIS
LIN {X 115.1035,Y 41.313,Z 136,A 16.1313,B 24.9468,C -1.6854,E1 25.1501,E2 429.976} C_DIS
LIN {X 113.9852,Y 44.3048,Z 136,A 17.6391,B 24.9464,C -1.6904,E1 25.1486,E2 428.4646} C_DIS
LIN {X 112.5172,Y 47.9153,Z 136,A 19.377,B 24.9464,C -1.6914,E1 25.1467,E2 426.7341} C_DIS
LIN {X 110.8369,Y 51.6805,Z 136,A 21.4794,B 24.9455,C -1.7056,E1 25.1442,E2 424.6096} C_DIS
LIN {X 109.0593,Y 55.3319,Z 136,A 23.2529,B 24.9455,C -1.7045,E1 25.1421,E2 422.8482} C_DIS
LIN {X 107.5335,Y 58.2465,Z 136,A 24.8419,B 24.9451,C -1.7112,E1 25.14,E2 421.2517} C_DIS
LIN {X 105.8235,Y 61.2975,Z 136,A 26.4818,B 24.9448,C -1.7157,E1 25.1377,E2 419.6096} C_DIS
LIN {X 103.6353,Y 64.9297,Z 136,A 28.5073,B 24.9444,C -1.723,E1 25.1347,E2 417.5772} C_DIS
LIN {X 101.3364,Y 68.4612,Z 136,A 30.4577,B 24.9441,C -1.727,E1 25.1317,E2 415.6271} C_DIS
LIN {X 98.8001,Y 72.074,Z 136,A 32.4961,B 24.9439,C -1.7308,E1 25.1284,E2 413.5897} C_DIS
LIN {X 96.3704,Y 75.2916,Z 136,A 34.4146,B 24.9435,C -1.7369,E1 25.1251,E2 411.6657} C_DIS
LIN {X 93.835,Y 78.4285,Z 136,A 36.2853,B 24.9432,C -1.7405,E1 25.1218,E2 409.7952} C_DIS
LIN {X 91.4307,Y 81.2185,Z 136,A 38.7915,B 24.9404,C -1.7835,E1 25.117,E2 407.1986} C_DIS
LIN {X 87.3589,Y 85.5828,Z 136,A 40.732,B 24.9428,C -1.747,E1 25.1134,E2 405.3527} C_DIS
LIN {X 84.3471,Y 88.5528,Z 136,A 42.6781,B 24.9426,C -1.7495,E1 25.1095,E2 403.4089} C_DIS
LIN {X 81.4078,Y 91.2623,Z 136,A 44.7061,B 24.9419,C -1.761,E1 25.1052,E2 401.3619} C_DIS
LIN {X 77.9399,Y 94.241,Z 136,A 47.6179,B 24.939,C -1.8033,E1 25.0988,E2 398.3612} C_DIS
LIN {X 72.9695,Y 98.14,Z 136,A 49.643,B 24.9418,C -1.7625,E1 25.0945,E2 396.44} C_DIS
LIN {X 69.8674,Y 100.372,Z 136,A 51.3738,B 24.9418,C -1.7627,E1 25.0906,E2 394.7147} C_DIS
LIN {X 66.9588,Y 102.3358,Z 136,A 53.1353,B 24.9412,C -1.7711,E1 25.0864,E2 392.9392} C_DIS
LIN {X 63.6274,Y 104.4398,Z 136,A 54.87,B 24.9414,C -1.7685,E1 25.0824,E2 391.2161} C_DIS
LIN {X 60.6134,Y 106.2168,Z 136,A 56.5145,B 24.9412,C -1.7712,E1 25.0784,E2 389.5702} C_DIS
LIN {X 57.58,Y 107.8919,Z 136,A 58.1065,B 24.9412,C -1.7719,E1 25.0745,E2 387.9811} C_DIS
LIN {X 54.4924,Y 109.482,Z 136,A 59.7777,B 24.9409,C -1.7762,E1 25.0703,E2 386.3043} C_DIS
LIN {X 51.2598,Y 111.0314,Z 136,A 61.4492,B 24.9408,C -1.7779,E1 25.0661,E2 384.6332} C_DIS
LIN {X 47.5551,Y 112.6688,Z 136,A 63.354,B 24.9406,C -1.7803,E1 25.0612,E2 382.7271} C_DIS
LIN {X 44.4683,Y 113.9217,Z 136,A 64.8665,B 24.9406,C -1.7796,E1 25.0573,E2 381.2197} C_DIS
LIN {X 41.2909,Y 115.1115,Z 136,A 66.4622,B 24.9406,C -1.7814,E1 25.0531,E2 379.6231} C_DIS
LIN {X 37.5223,Y 116.3948,Z 136,A 68.321,B 24.9404,C -1.7827,E1 25.0482,E2 377.7649} C_DIS
LIN {X 34.1434,Y 117.4302,Z 136,A 69.8554,B 24.9407,C -1.7781,E1 25.0441,E2 376.2439} C_DIS
LIN {X 30.0781,Y 118.5365,Z 136,A 71.9569,B 24.9402,C -1.7855,E1 25.0384,E2 374.1284} C_DIS
LIN {X 26.4504,Y 119.4002,Z 136,A 73.7668,B 24.94,C -1.7894,E1 25.0334,E2 372.3116} C_DIS
LIN {X 22.7258,Y 120.1632,Z 136,A 75.4005,B 24.9404,C -1.7832,E1 25.029,E2 370.6946} C_DIS
LIN {X 18.4577,Y 120.8925,Z 136,A 77.4461,B 24.9404,C -1.7847,E1 25.0234,E2 368.6476} C_DIS
LIN {X 11.8039,Y 121.7223,Z 136,A 80.6179,B 24.9402,C -1.7866,E1 25.0146,E2 365.4734} C_DIS
LIN {X 8.2936,Y 122.0133,Z 136,A 82.4066,B 24.9397,C -1.7932,E1 25.0096,E2 363.6701} C_DIS
LIN {X 4.2023,Y 122.2224,Z 136,A 84.301,B 24.9398,C -1.7919,E1 25.0043,E2 361.7792} C_DIS
LIN {X 0.2564,Y 122.2938,Z 136,A 86.09,B 24.94,C -1.7888,E1 24.9993,E2 359.9978} C_DIS
LIN {X -3.3062,Y 122.2487,Z 136,A 87.7328,B 24.9401,C -1.7871,E1 24.9947,E2 358.3587} C_DIS
LIN {X -7.3247,Y 122.0739,Z 136,A 89.6144,B 24.9401,C -1.7863,E1 24.9895,E2 356.4786} C_DIS
LIN {X -11.1387,Y 121.7862,Z 136,A 91.2709,B 24.9407,C -1.7792,E1 24.9849,E2 354.8383} C_DIS
LIN {X -14.8456,Y 121.3893,Z 136,A 92.8677,B 24.9412,C -1.7713,E1 24.9805,E2 353.2591} C_DIS
LIN {X -22.2053,Y 120.2622,Z 136,A 96.5783,B 24.9407,C -1.7789,E1 24.9703,E2 349.5271} C_DIS
LIN {X -28.0304,Y 119.0391,Z 136,A 99.7819,B 24.9396,C -1.7955,E1 24.9614,E2 346.2802} C_DIS
LIN {X -31.1825,Y 118.2512,Z 136,A 101.0996,B 24.9403,C -1.7846,E1 24.9579,E2 344.9865} C_DIS
LIN {X -35.514,Y 117.0231,Z 136,A 103.1053,B 24.9408,C -1.7775,E1 24.9526,E2 342.9943} C_DIS
LIN {X -38.9068,Y 115.9392,Z 136,A 104.7101,B 24.9411,C -1.7726,E1 24.9483,E2 341.3983} C_DIS
LIN {X -42.5265,Y 114.6613,Z 136,A 106.5838,B 24.9411,C -1.7737,E1 24.9434,E2 339.5182} C_DIS
LIN {X -45.62,Y 113.4653,Z 136,A 108.3336,B 24.9406,C -1.7804,E1 24.9388,E2 337.7486} C_DIS
LIN {X -49.9133,Y 111.6432,Z 136,A 110.3196,B 24.9414,C -1.7681,E1 24.9338,E2 335.7871} C_DIS
LIN {X -53.2351,Y 110.0994,Z 136,A 111.9952,B 24.9417,C -1.7636,E1 24.9296,E2 334.1181} C_DIS
LIN {X -56.7624,Y 108.3216,Z 136,A 113.7858,B 24.9421,C -1.7578,E1 24.9251,E2 332.3364} C_DIS
LIN {X -60.124,Y 106.4948,Z 136,A 115.4914,B 24.9426,C -1.7507,E1 24.921,E2 330.6427} C_DIS
LIN {X -63.7617,Y 104.3575,Z 136,A 117.6354,B 24.9423,C -1.7545,E1 24.9158,E2 328.4831} C_DIS
LIN {X -68.4764,Y 101.3261,Z 136,A 120.8597,B 24.9409,C -1.7763,E1 24.9081,E2 325.1965} C_DIS
LIN {X -72.0421,Y 98.8232,Z 136,A 122.4698,B 24.9424,C -1.7527,E1 24.9046,E2 323.6369} C_DIS
LIN {X -74.8305,Y 96.7285,Z 136,A 124.1381,B 24.9426,C -1.7507,E1 24.9009,E2 321.9673} C_DIS
LIN {X -78.3578,Y 93.8943,Z 136,A 126.2254,B 24.943,C -1.7445,E1 24.8964,E2 319.8869} C_DIS
LIN {X -81.1518,Y 91.49,Z 136,A 127.9782,B 24.9432,C -1.7417,E1 24.8927,E2 318.1339} C_DIS
LIN {X -84.3751,Y 88.526,Z 136,A 130.1123,B 24.9432,C -1.7404,E1 24.8884,E2 315.9939} C_DIS
LIN {X -87.6339,Y 85.3017,Z 136,A 132.1963,B 24.9438,C -1.7323,E1 24.8843,E2 313.9204} C_DIS
LIN {X -90.8732,Y 81.8422,Z 136,A 134.427,B 24.9441,C -1.7271,E1 24.8801,E2 311.6923} C_DIS
LIN {X -94.0204,Y 78.2063,Z 136,A 136.6485,B 24.9446,C -1.7198,E1 24.8761,E2 309.478} C_DIS
LIN {X -96.4565,Y 75.1814,Z 136,A 138.5113,B 24.9448,C -1.7168,E1 24.8729,E2 307.6137} C_DIS
LIN {X -99.1506,Y 71.5904,Z 136,A 140.544,B 24.9453,C -1.7079,E1 24.8695,E2 305.5924} C_DIS
LIN {X -102.9309,Y 66.0395,Z 136,A 143.7437,B 24.9458,C -1.7013,E1 24.8646,E2 302.3924} C_DIS
LIN {X -105.0175,Y 62.6682,Z 136,A 145.5895,B 24.9461,C -1.6954,E1 24.8619,E2 300.5512} C_DIS
LIN {X -106.9672,Y 59.2791,Z 136,A 147.4353,B 24.9464,C -1.6906,E1 24.8593,E2 298.7071} C_DIS
LIN {X -108.2094,Y 56.9761,Z 136,A 149.204,B 24.9451,C -1.7108,E1 24.857,E2 296.8807} C_DIS
LIN {X -110.188,Y 53.0498,Z 136,A 150.7078,B 24.9471,C -1.6801,E1 24.8552,E2 295.4421} C_DIS
LIN {X -111.6491,Y 49.9,Z 136,A 152.3401,B 24.9474,C -1.6754,E1 24.8533,E2 293.8122} C_DIS
LIN {X -113.0529,Y 46.6355,Z 136,A 153.9572,B 24.9479,C -1.6681,E1 24.8516,E2 292.2034} C_DIS
LIN {X -114.5124,Y 42.9239,Z 136,A 155.892,B 24.948,C -1.6651,E1 24.8496,E2 290.2647} C_DIS
LIN {X -115.5994,Y 39.9046,Z 136,A 158.6427,B 24.9449,C -1.7154,E1 24.8471,E2 287.3785} C_DIS
LIN {X -117.8195,Y 32.7746,Z 136,A 160.961,B 24.9489,C -1.652,E1 24.8454,E2 285.198} C_DIS
LIN {X -118.8388,Y 28.8611,Z 136,A 162.8558,B 24.9492,C -1.6459,E1 24.8441,E2 283.3067} C_DIS
LIN {X -120.029,Y 23.4281,Z 136,A 165.52,B 24.9496,C -1.64,E1 24.8425,E2 280.6409} C_DIS
LIN {X -120.6029,Y 20.2628,Z 136,A 167.017,B 24.9499,C -1.6346,E1 24.8418,E2 279.1478} C_DIS
LIN {X -121.0411,Y 17.4553,Z 136,A 168.416,B 24.95,C -1.6332,E1 24.8412,E2 277.7438} C_DIS
LIN {X -121.579,Y 13.1979,Z 136,A 170.2621,B 24.9509,C -1.6195,E1 24.8406,E2 275.9195} C_DIS
LIN {X -121.9576,Y 9.056,Z 136,A 172.3628,B 24.9509,C -1.6197,E1 24.8401,E2 273.8056} C_DIS
LIN {X -122.1957,Y 4.8863,Z 136,A 174.5027,B 24.9507,C -1.6213,E1 24.8399,E2 271.649} C_DIS
LIN {X -122.2774,Y -1.9791,Z 136,A 177.5259,B 24.9519,C -1.6022,E1 24.8399,E2 268.653} C_DIS
LIN {X -122.1597,Y -5.729,Z 136,A 179.1219,B 24.9527,C -1.5894,E1 24.8399,E2 267.0779} C_DIS
LIN {X -121.8014,Y -10.9788,Z 136,A -178.1205,B 24.9524,C -1.5941,E1 24.8406,E2 264.2925} C_DIS
LIN {X -121.275,Y -15.7488,Z 136,A -175.9524,B 24.953,C -1.5834,E1 24.8413,E2 262.1371} C_DIS
LIN {X -120.7529,Y -19.359,Z 136,A -174.0991,B 24.953,C -1.5842,E1 24.8421,E2 260.2708} C_DIS
LIN {X -120.179,Y -22.6431,Z 136,A -172.4441,B 24.953,C -1.5833,E1 24.8429,E2 258.608} C_DIS
LIN {X -119.2559,Y -27.086,Z 136,A -170.5956,B 24.9541,C -1.5645,E1 24.844,E2 256.7937} C_DIS
LIN {X -118.5361,Y -30.0797,Z 136,A -169.0384,B 24.9541,C -1.565,E1 24.845,E2 255.2261} C_DIS
LIN {X -117.4557,Y -34.0563,Z 136,A -167.1017,B 24.9544,C -1.5592,E1 24.8465,E2 253.2919} C_DIS
LIN {X -116.4736,Y -37.2755,Z 136,A -165.5394,B 24.9548,C -1.5538,E1 24.8478,E2 251.7336} C_DIS
LIN {X -115.313,Y -40.7305,Z 136,A -163.5013,B 24.9542,C -1.5632,E1 24.8497,E2 249.6615} C_DIS
LIN {X -113.4696,Y -45.6093,Z 136,A -161.3645,B 24.9554,C -1.5424,E1 24.8518,E2 247.5623} C_DIS
LIN {X -112.2635,Y -48.5021,Z 136,A -159.9965,B 24.9559,C -1.5337,E1 24.8533,E2 246.2075} C_DIS
LIN {X -110.4671,Y -52.4656,Z 136,A -157.8136,B 24.9559,C -1.5341,E1 24.8559,E2 244.0116} C_DIS
LIN {X -109.116,Y -55.2205,Z 136,A -156.5453,B 24.9566,C -1.5226,E1 24.8574,E2 242.764} C_DIS
LIN {X -107.6828,Y -57.969,Z 136,A -154.8902,B 24.9563,C -1.5275,E1 24.8596,E2 241.0884} C_DIS
LIN {X -105.3543,Y -62.1006,Z 136,A -152.6419,B 24.9566,C -1.5225,E1 24.8627,E2 238.8401} C_DIS
LIN {X -103.2306,Y -65.5709,Z 136,A -150.4195,B 24.9561,C -1.5316,E1 24.8661,E2 236.5849} C_DIS
LIN {X -101.41,Y -68.3524,Z 136,A -149.1074,B 24.9569,C -1.5166,E1 24.8681,E2 235.302} C_DIS
LIN {X -98.855,Y -71.9982,Z 136,A -146.9834,B 24.9571,C -1.513,E1 24.8715,E2 233.1762} C_DIS
LIN {X -96.7966,Y -74.7426,Z 136,A -145.2232,B 24.9569,C -1.5159,E1 24.8746,E2 231.4007} C_DIS
LIN {X -93.508,Y -78.8183,Z 136,A -142.9438,B 24.9577,C -1.5022,E1 24.8786,E2 229.1434} C_DIS
LIN {X -91.198,Y -81.4796,Z 136,A -141.0773,B 24.9574,C -1.5081,E1 24.8821,E2 227.2544} C_DIS
LIN {X -87.5927,Y -85.3444,Z 136,A -138.9011,B 24.9585,C -1.489,E1 24.8862,E2 225.1142} C_DIS
LIN {X -83.554,Y -89.3018,Z 136,A -136.0957,B 24.9584,C -1.4905,E1 24.8919,E2 222.2936} C_DIS
LIN {X -80.1707,Y -92.3512,Z 136,A -134.1188,B 24.959,C -1.4791,E1 24.8959,E2 220.3361} C_DIS
LIN {X -75.6853,Y -96.0612,Z 136,A -131.2679,B 24.959,C -1.4795,E1 24.9022,E2 217.4733} C_DIS
LIN {X -72.5812,Y -98.4277,Z 136,A -129.4073,B 24.959,C -1.4777,E1 24.9063,E2 215.6103} C_DIS
LIN {X -69.3086,Y -100.7587,Z 136,A -127.4403,B 24.959,C -1.4784,E1 24.9108,E2 213.635} C_DIS
LIN {X -65.6693,Y -103.1678,Z 136,A -124.8209,B 24.9578,C -1.5017,E1 24.9172,E2 210.9518} C_DIS
LIN {X -61.2589,Y -105.8458,Z 136,A -123.101,B 24.9597,C -1.4659,E1 24.9211,E2 209.3119} C_DIS
LIN {X -57.6962,Y -107.8294,Z 136,A -121.16,B 24.9598,C -1.4647,E1 24.9259,E2 207.3682} C_DIS
LIN {X -54.5575,Y -109.4498,Z 136,A -119.5035,B 24.9599,C -1.4626,E1 24.93,E2 205.7121} C_DIS
LIN {X -51.5067,Y -110.9173,Z 136,A -117.9861,B 24.9602,C -1.4576,E1 24.9338,E2 204.2029} C_DIS
LIN {X -48.2158,Y -112.3873,Z 136,A -116.095,B 24.9598,C -1.4651,E1 24.9387,E2 202.2895} C_DIS
LIN {X -44.2839,Y -113.9934,Z 136,A -114.2253,B 24.9602,C -1.4575,E1 24.9435,E2 200.4336} C_DIS
LIN {X -40.4319,Y -115.4165,Z 136,A -112.3425,B 24.9604,C -1.4539,E1 24.9484,E2 198.5558} C_DIS
LIN {X -37.086,Y -116.5342,Z 136,A -110.815,B 24.9608,C -1.4467,E1 24.9525,E2 197.0424} C_DIS
LIN {X -32.9812,Y -117.7617,Z 136,A -108.6726,B 24.9605,C -1.4516,E1 24.9582,E2 194.8849} C_DIS
LIN {X -29.5623,Y -118.6674,Z 136,A -106.918,B 24.9603,C -1.4552,E1 24.963,E2 193.1192} C_DIS
LIN {X -26.1379,Y -119.4677,Z 136,A -105.462,B 24.9609,C -1.4454,E1 24.9669,E2 191.6847} C_DIS
LIN {X -21.6648,Y -120.3589,Z 136,A -103.2437,B 24.9607,C -1.4484,E1 24.973,E2 189.4569} C_DIS
LIN {X -18.9835,Y -120.8111,Z 136,A -101.5579,B 24.9597,C -1.4675,E1 24.9778,E2 187.7241} C_DIS
LIN {X -15.3417,Y -121.3283,Z 136,A -100.2463,B 24.9607,C -1.4476,E1 24.9813,E2 186.4588} C_DIS
LIN {X -11.9965,Y -121.7038,Z 136,A -98.5832,B 24.9605,C -1.4515,E1 24.986,E2 184.7854} C_DIS
LIN {X -7.7456,Y -122.048,Z 136,A -96.655,B 24.9607,C -1.4482,E1 24.9913,E2 182.8644} C_DIS
LIN {X -4.3027,Y -122.2185,Z 136,A -95.0653,B 24.9607,C -1.4471,E1 24.9957,E2 181.2769} C_DIS
LIN {X -0.7213,Y -122.2913,Z 136,A -93.3569,B 24.9607,C -1.4489,E1 25.0005,E2 179.5643} C_DIS
LIN {X -0.7213,Y -122.2913,Z 136,A -93.3569,B 24.9607,C -1.4489,E1 25.0005,E2 179.5643} C_DIS
Enddeposition()
LIN {X 0.8685,Y -121.3008,Z 136,A -93.3868,B 24.9617,C -1.4297,E1 25.0003,E2 179.6395} C_DIS
Startdeposition()
$VEL.CP = VEL_PRINT
LIN {X -2.3665,Y -121.2812,Z 136,A -94.9952,B 24.9619,C -1.4257,E1 24.9958,E2 181.2576} C_DIS
LIN {X -5.8455,Y -121.163,Z 136,A -96.5279,B 24.9617,C -1.4307,E1 24.9916,E2 182.7787} C_DIS
LIN {X -9.5444,Y -120.9294,Z 136,A -98.4713,B 24.9621,C -1.4217,E1 24.9861,E2 184.7441} C_DIS
LIN {X -14.0701,Y -120.4852,Z 136,A -100.4782,B 24.9618,C -1.4285,E1 24.9805,E2 186.7361} C_DIS
LIN {X -17.8574,Y -119.984,Z 136,A -102.2057,B 24.9616,C -1.4325,E1 24.9758,E2 188.4555} C_DIS
LIN {X -20.7276,Y -119.5213,Z 136,A -103.7644,B 24.962,C -1.4244,E1 24.9714,E2 190.035} C_DIS
LIN {X -24.5523,Y -118.7933,Z 136,A -105.5461,B 24.9618,C -1.4278,E1 24.9666,E2 191.8106} C_DIS
LIN {X -28.635,Y -117.8754,Z 136,A -107.431,B 24.9615,C -1.433,E1 24.9615,E2 193.6856} C_DIS
LIN {X -31.7635,Y -117.0721,Z 136,A -108.9257,B 24.9615,C -1.4353,E1 24.9575,E2 195.177} C_DIS
LIN {X -35.222,Y -116.0776,Z 136,A -110.7943,B 24.9618,C -1.4289,E1 24.9524,E2 197.0641} C_DIS
LIN {X -38.889,Y -114.9021,Z 136,A -112.4539,B 24.9613,C -1.4376,E1 24.948,E2 198.7061} C_DIS
LIN {X -41.6922,Y -113.9148,Z 136,A -113.8467,B 24.9612,C -1.4393,E1 24.9444,E2 200.0975} C_DIS
LIN {X -44.4717,Y -112.8586,Z 136,A -115.2703,B 24.9612,C -1.4398,E1 24.9407,E2 201.523} C_DIS
LIN {X -47.4797,Y -111.6274,Z 136,A -116.9356,B 24.9614,C -1.4355,E1 24.9363,E2 203.2023} C_DIS
LIN {X -51.0852,Y -110.0219,Z 136,A -118.7139,B 24.9611,C -1.4416,E1 24.9318,E2 204.9705} C_DIS
LIN {X -54.0013,Y -108.6208,Z 136,A -120.2112,B 24.9609,C -1.4448,E1 24.9281,E2 206.464} C_DIS
LIN {X -56.6458,Y -107.2651,Z 136,A -121.6314,B 24.9609,C -1.4459,E1 24.9246,E2 207.8855} C_DIS
LIN {X -59.7909,Y -105.5467,Z 136,A -123.4697,B 24.9611,C -1.4417,E1 24.9201,E2 209.7391} C_DIS
LIN {X -63.1678,Y -103.5608,Z 136,A -125.1585,B 24.9605,C -1.4517,E1 24.9161,E2 211.4094} C_DIS
LIN {X -66.2629,Y -101.6081,Z 136,A -127.0138,B 24.9607,C -1.4488,E1 24.9117,E2 213.2776} C_DIS
LIN {X -69.3555,Y -99.5226,Z 136,A -128.7994,B 24.9606,C -1.4506,E1 24.9075,E2 215.0647} C_DIS
LIN {X -72.2636,Y -97.4317,Z 136,A -130.3592,B 24.9601,C -1.4595,E1 24.9041,E2 216.609} C_DIS
LIN {X -75.245,Y -95.1485,Z 136,A -132.313,B 24.9604,C -1.4547,E1 24.8997,E2 218.5813} C_DIS
LIN {X -78.3462,Y -92.6114,Z 136,A -134.2027,B 24.9602,C -1.4585,E1 24.8957,E2 220.4692} C_DIS
LIN {X -81.4612,Y -89.8832,Z 136,A -136.0765,B 24.9597,C -1.466,E1 24.8918,E2 222.3325} C_DIS
LIN {X -84.1684,Y -87.3538,Z 136,A -137.9252,B 24.9597,C -1.4654,E1 24.888,E2 224.1905} C_DIS
LIN {X -87.0317,Y -84.5011,Z 136,A -139.8316,B 24.9595,C -1.4696,E1 24.8843,E2 226.0948} C_DIS
LIN {X -89.6014,Y -81.7718,Z 136,A -141.575,B 24.9593,C -1.4748,E1 24.881,E2 227.8336} C_DIS
LIN {X -92.1434,Y -78.8964,Z 136,A -143.3653,B 24.959,C -1.48,E1 24.8777,E2 229.6196} C_DIS
LIN {X -94.7028,Y -75.805,Z 136,A -145.3587,B 24.959,C -1.4803,E1 24.8742,E2 231.6215} C_DIS
LIN {X -97.4349,Y -72.2594,Z 136,A -147.3261,B 24.9583,C -1.4919,E1 24.8709,E2 233.5707} C_DIS
LIN {X -99.3693,Y -69.5757,Z 136,A -149.0222,B 24.9584,C -1.4901,E1 24.8681,E2 235.2794} C_DIS
LIN {X -101.689,Y -66.1382,Z 136,A -150.8592,B 24.9578,C -1.5005,E1 24.8653,E2 237.1009} C_DIS
LIN {X -103.5951,Y -63.1119,Z 136,A -152.6293,B 24.9578,C -1.5015,E1 24.8627,E2 238.8777} C_DIS
LIN {X -105.2357,Y -60.336,Z 136,A -154.0961,B 24.9574,C -1.508,E1 24.8606,E2 240.3365} C_DIS
LIN {X -106.693,Y -57.7203,Z 136,A -155.6708,B 24.9576,C -1.505,E1 24.8585,E2 241.9267} C_DIS
LIN {X -108.3513,Y -54.5414,Z 136,A -157.3287,B 24.9572,C -1.5113,E1 24.8564,E2 243.5783} C_DIS
LIN {X -110.0368,Y -51.0528,Z 136,A -159.0589,B 24.9567,C -1.5209,E1 24.8543,E2 245.2951} C_DIS
LIN {X -111.4207,Y -47.9576,Z 136,A -160.7012,B 24.9565,C -1.5238,E1 24.8525,E2 246.9396} C_DIS
LIN {X -112.8553,Y -44.4801,Z 136,A -162.6703,B 24.9567,C -1.5208,E1 24.8504,E2 248.9269} C_DIS
LIN {X -114.2074,Y -40.8808,Z 136,A -164.2922,B 24.9559,C -1.5346,E1 24.8489,E2 250.5251} C_DIS
LIN {X -115.3725,Y -37.4705,Z 136,A -166.1515,B 24.9559,C -1.533,E1 24.8472,E2 252.3988} C_DIS
LIN {X -116.4541,Y -33.9553,Z 136,A -167.7784,B 24.9554,C -1.5431,E1 24.8459,E2 254.011} C_DIS
LIN {X -117.4539,Y -30.3208,Z 136,A -169.6248,B 24.9552,C -1.5458,E1 24.8446,E2 255.8617} C_DIS
LIN {X -118.3562,Y -26.5808,Z 136,A -171.5117,B 24.9551,C -1.5485,E1 24.8434,E2 257.7532} C_DIS
LIN {X -119.1428,Y -22.7931,Z 136,A -173.2123,B 24.9544,C -1.5597,E1 24.8425,E2 259.4371} C_DIS
LIN {X -119.7468,Y -19.3805,Z 136,A -174.876,B 24.9542,C -1.5638,E1 24.8417,E2 261.101} C_DIS
LIN {X -120.201,Y -16.3277,Z 136,A -176.3336,B 24.9539,C -1.5685,E1 24.8411,E2 262.5562} C_DIS
LIN {X -120.5658,Y -13.3644,Z 136,A -177.8851,B 24.9539,C -1.567,E1 24.8406,E2 264.1203} C_DIS
LIN {X -120.9327,Y -9.5028,Z 136,A -179.7678,B 24.9538,C -1.5708,E1 24.8402,E2 266.0054} C_DIS
LIN {X -121.1755,Y -5.5963,Z 136,A 178.4129,B 24.9533,C -1.5781,E1 24.8399,E2 267.8183} C_DIS
LIN {X -121.2956,Y -1.5018,Z 136,A 176.617,B 24.9526,C -1.5903,E1 24.8398,E2 269.5959} C_DIS
LIN {X -121.2963,Y 1.4599,Z 136,A 175.2659,B 24.9522,C -1.5969,E1 24.8398,E2 270.9393} C_DIS
LIN {X -121.2215,Y 4.4725,Z 136,A 173.7461,B 24.9522,C -1.5975,E1 24.8399,E2 272.4669} C_DIS
LIN {X -121.0754,Y 7.4383,Z 136,A 172.2579,B 24.9522,C -1.5985,E1 24.8402,E2 273.9617} C_DIS
LIN {X -120.7194,Y 11.895,Z 136,A 170.0884,B 24.9519,C -1.6029,E1 24.8407,E2 276.1336} C_DIS
LIN {X -120.2816,Y 15.7127,Z 136,A 168.3816,B 24.9512,C -1.6135,E1 24.8413,E2 277.8254} C_DIS
LIN {X -119.7646,Y 19.2736,Z 136,A 166.6628,B 24.9509,C -1.6182,E1 24.842,E2 279.5432} C_DIS
LIN {X -119.1416,Y 22.7996,Z 136,A 164.9281,B 24.9507,C -1.6219,E1 24.8429,E2 281.2794} C_DIS
LIN {X -118.5431,Y 25.731,Z 136,A 163.5124,B 24.9504,C -1.6264,E1 24.8437,E2 282.6929} C_DIS
LIN {X -117.6682,Y 29.4763,Z 136,A 161.5833,B 24.9504,C -1.6275,E1 24.8449,E2 284.6306} C_DIS
LIN {X -116.597,Y 33.4672,Z 136,A 159.6201,B 24.95,C -1.6332,E1 24.8464,E2 286.5914} C_DIS
LIN {X -115.349,Y 37.5441,Z 136,A 157.7262,B 24.9493,C -1.6447,E1 24.848,E2 288.4689} C_DIS
LIN {X -114.4113,Y 40.3103,Z 136,A 156.3358,B 24.9491,C -1.6486,E1 24.8492,E2 289.8579} C_DIS
LIN {X -113.4934,Y 42.8232,Z 136,A 155.03,B 24.9489,C -1.6508,E1 24.8505,E2 291.1658} C_DIS
LIN {X -112.2999,Y 45.864,Z 136,A 153.5071,B 24.9486,C -1.6565,E1 24.8521,E2 292.6838} C_DIS
LIN {X -110.8963,Y 49.1594,Z 136,A 151.8115,B 24.9483,C -1.6615,E1 24.854,E2 294.3765} C_DIS
LIN {X -109.5249,Y 52.1421,Z 136,A 150.1312,B 24.9483,C -1.6608,E1 24.856,E2 296.0679} C_DIS
LIN {X -107.944,Y 55.3415,Z 136,A 148.5463,B 24.9477,C -1.6701,E1 24.8579,E2 297.639} C_DIS
LIN {X -106.4879,Y 58.0968,Z 136,A 146.9853,B 24.9477,C -1.6707,E1 24.86,E2 299.2069} C_DIS
LIN {X -104.5848,Y 61.4567,Z 136,A 145.1572,B 24.9474,C -1.6759,E1 24.8626,E2 301.0322} C_DIS
LIN {X -102.8212,Y 64.3648,Z 136,A 143.4757,B 24.9473,C -1.6773,E1 24.865,E2 302.7189} C_DIS
LIN {X -100.5414,Y 67.8702,Z 136,A 141.5724,B 24.9467,C -1.686,E1 24.8679,E2 304.6111} C_DIS
LIN {X -98.7122,Y 70.504,Z 136,A 139.9604,B 24.9467,C -1.686,E1 24.8706,E2 306.2308} C_DIS
LIN {X -96.0837,Y 74.0469,Z 136,A 137.9042,B 24.9463,C -1.6929,E1 24.874,E2 308.2805} C_DIS
LIN {X -93.5784,Y 77.1884,Z 136,A 135.9497,B 24.9461,C -1.6955,E1 24.8774,E2 310.2378} C_DIS
LIN {X -90.7277,Y 80.5199,Z 136,A 133.8639,B 24.9458,C -1.7003,E1 24.8813,E2 312.3217} C_DIS
LIN {X -87.8518,Y 83.6483,Z 136,A 131.8489,B 24.9455,C -1.705,E1 24.8851,E2 314.3342} C_DIS
LIN {X -84.7231,Y 86.8159,Z 136,A 129.8141,B 24.945,C -1.7131,E1 24.8891,E2 316.3584} C_DIS
LIN {X -81.9207,Y 89.4649,Z 136,A 127.9154,B 24.945,C -1.7141,E1 24.893,E2 318.2625} C_DIS
LIN {X -78.899,Y 92.1411,Z 136,A 126.0652,B 24.9445,C -1.7209,E1 24.8969,E2 320.1037} C_DIS
LIN {X -75.8051,Y 94.7027,Z 136,A 124.1625,B 24.9442,C -1.7249,E1 24.901,E2 322.0042} C_DIS
LIN {X -72.7569,Y 97.0644,Z 136,A 122.2451,B 24.9442,C -1.7246,E1 24.9053,E2 323.9291} C_DIS
LIN {X -69.2912,Y 99.5673,Z 136,A 120.3257,B 24.9437,C -1.7332,E1 24.9096,E2 325.8349} C_DIS
LIN {X -66.1332,Y 101.6923,Z 136,A 118.5733,B 24.9433,C -1.7387,E1 24.9137,E2 327.5799} C_DIS
LIN {X -63.6333,Y 103.2752,Z 136,A 117.0558,B 24.9435,C -1.7361,E1 24.9173,E2 329.1084} C_DIS
LIN {X -60.3073,Y 105.2521,Z 136,A 115.3359,B 24.943,C -1.7441,E1 24.9214,E2 330.8143} C_DIS
LIN {X -57.7125,Y 106.6973,Z 136,A 113.7714,B 24.9433,C -1.7395,E1 24.9253,E2 332.3943} C_DIS
LIN {X -54.538,Y 108.353,Z 136,A 112.081,B 24.9431,C -1.7424,E1 24.9295,E2 334.0825} C_DIS
LIN {X -51.0746,Y 110.0268,Z 136,A 110.4053,B 24.9425,C -1.7515,E1 24.9336,E2 335.7408} C_DIS
LIN {X -47.8005,Y 111.4887,Z 136,A 108.593,B 24.9427,C -1.7487,E1 24.9383,E2 337.5639} C_DIS
LIN {X -43.8607,Y 113.0961,Z 136,A 106.7193,B 24.9421,C -1.7576,E1 24.9431,E2 339.4206} C_DIS
LIN {X -40.855,Y 114.2167,Z 136,A 105.1681,B 24.9421,C -1.758,E1 24.9472,E2 340.9741} C_DIS
LIN {X -37.46,Y 115.3758,Z 136,A 103.3852,B 24.9422,C -1.7561,E1 24.9519,E2 342.7648} C_DIS
LIN {X -33.785,Y 116.504,Z 136,A 101.6314,B 24.9419,C -1.7609,E1 24.9566,E2 344.5101} C_DIS
LIN {X -30.1946,Y 117.4859,Z 136,A 99.8267,B 24.9419,C -1.7607,E1 24.9615,E2 346.3182} C_DIS
LIN {X -26.5383,Y 118.3659,Z 136,A 97.9661,B 24.942,C -1.7585,E1 24.9666,E2 348.1862} C_DIS
LIN {X -22.7998,Y 119.1416,Z 136,A 96.3034,B 24.9415,C -1.7664,E1 24.9711,E2 349.8322} C_DIS
LIN {X -19.2385,Y 119.7702,Z 136,A 94.5384,B 24.9416,C -1.765,E1 24.9759,E2 351.6021} C_DIS
LIN {X -15.705,Y 120.2826,Z 136,A 92.8791,B 24.9415,C -1.7674,E1 24.9805,E2 353.2571} C_DIS
LIN {X -12.4967,Y 120.6592,Z 136,A 91.2236,B 24.9418,C -1.7623,E1 24.9852,E2 354.9255} C_DIS
LIN {X -8.7153,Y 120.9902,Z 136,A 89.5341,B 24.9414,C -1.7679,E1 24.9898,E2 356.6027} C_DIS
LIN {X -5.0655,Y 121.1984,Z 136,A 87.8409,B 24.9413,C -1.77,E1 24.9945,E2 358.2913} C_DIS
LIN {X -1.4846,Y 121.2958,Z 136,A 86.181,B 24.9412,C -1.7719,E1 24.9992,E2 359.9469} C_DIS
LIN {X 1.4883,Y 121.2958,Z 136,A 84.5642,B 24.9418,C -1.7624,E1 25.0037,E2 361.5859} C_DIS
LIN {X 5.9587,Y 121.1573,Z 136,A 82.6363,B 24.9412,C -1.771,E1 25.0091,E2 363.493} C_DIS
LIN {X 8.9265,Y 120.9748,Z 136,A 81.2387,B 24.9412,C -1.7713,E1 25.0129,E2 364.8893} C_DIS
LIN {X 11.9335,Y 120.7157,Z 136,A 79.8205,B 24.9412,C -1.7715,E1 25.0169,E2 366.3062} C_DIS
LIN {X 14.8674,Y 120.3901,Z 136,A 78.4284,B 24.9412,C -1.7713,E1 25.0207,E2 367.6976} C_DIS
LIN {X 17.6167,Y 120.0184,Z 136,A 77.089,B 24.9413,C -1.7696,E1 25.0245,E2 369.0399} C_DIS
LIN {X 20.7638,Y 119.5148,Z 136,A 75.4337,B 24.9418,C -1.7622,E1 25.0291,E2 370.7111} C_DIS
LIN {X 24.5384,Y 118.7962,Z 136,A 73.6655,B 24.9418,C -1.7636,E1 25.0339,E2 372.4739} C_DIS
LIN {X 28.625,Y 117.8778,Z 136,A 71.7813,B 24.9415,C -1.7668,E1 25.039,E2 374.3478} C_DIS
LIN {X 31.7778,Y 117.0683,Z 136,A 70.2798,B 24.9415,C -1.7675,E1 25.043,E2 375.8453} C_DIS
LIN {X 35.2178,Y 116.0788,Z 136,A 68.4533,B 24.9419,C -1.76,E1 25.048,E2 377.6866} C_DIS
LIN {X 38.884,Y 114.9038,Z 136,A 66.7727,B 24.9416,C -1.7649,E1 25.0524,E2 379.3523} C_DIS
LIN {X 42.2624,Y 113.7035,Z 136,A 64.9169,B 24.9422,C -1.7557,E1 25.0573,E2 381.226} C_DIS
LIN {X 45.8448,Y 112.3077,Z 136,A 63.2776,B 24.9418,C -1.7621,E1 25.0615,E2 382.8465} C_DIS
LIN {X 49.1678,Y 110.8926,Z 136,A 61.4263,B 24.9424,C -1.7534,E1 25.0663,E2 384.714} C_DIS
LIN {X 52.6629,Y 109.2761,Z 136,A 59.7505,B 24.9421,C -1.7579,E1 25.0705,E2 386.3747} C_DIS
LIN {X 55.867,Y 107.674,Z 136,A 57.9252,B 24.9426,C -1.7494,E1 25.0751,E2 388.2153} C_DIS
LIN {X 59.7862,Y 105.5494,Z 136,A 55.9663,B 24.9424,C -1.7533,E1 25.0798,E2 390.1591} C_DIS
LIN {X 62.3538,Y 104.0529,Z 136,A 54.5439,B 24.9426,C -1.7503,E1 25.0832,E2 391.5841} C_DIS
LIN {X 65.65,Y 102.0053,Z 136,A 52.7369,B 24.9426,C -1.7487,E1 25.0875,E2 393.3893} C_DIS
LIN {X 68.6311,Y 100.0235,Z 136,A 51.0585,B 24.9428,C -1.7465,E1 25.0914,E2 395.0673} C_DIS
LIN {X 71.4993,Y 97.9944,Z 136,A 49.28,B 24.9434,C -1.7379,E1 25.0955,E2 396.8598} C_DIS
LIN {X 74.6944,Y 95.5811,Z 136,A 47.4244,B 24.9435,C -1.7361,E1 25.0996,E2 398.7128} C_DIS
LIN {X 77.7772,Y 93.0897,Z 136,A 45.5609,B 24.9437,C -1.7329,E1 25.1036,E2 400.5768} C_DIS
LIN {X 80.685,Y 90.5812,Z 136,A 43.692,B 24.9441,C -1.7266,E1 25.1075,E2 402.4531} C_DIS
LIN {X 83.9588,Y 87.5549,Z 136,A 41.6601,B 24.9441,C -1.7258,E1 25.1116,E2 404.4788} C_DIS
LIN {X 86.9058,Y 84.6311,Z 136,A 39.7345,B 24.9444,C -1.7232,E1 25.1154,E2 406.4023} C_DIS
LIN {X 89.6133,Y 81.7587,Z 136,A 37.8463,B 24.9447,C -1.7178,E1 25.119,E2 408.2948} C_DIS
LIN {X 92.0809,Y 78.9689,Z 136,A 36.1066,B 24.9449,C -1.7146,E1 25.1222,E2 410.0342} C_DIS
LIN {X 94.7105,Y 75.7953,Z 136,A 34.1826,B 24.9451,C -1.711,E1 25.1256,E2 411.9578} C_DIS
LIN {X 97.0536,Y 72.7713,Z 136,A 32.3147,B 24.9456,C -1.7036,E1 25.1288,E2 413.8345} C_DIS
LIN {X 99.5254,Y 69.3514,Z 136,A 30.4238,B 24.9456,C -1.7035,E1 25.1318,E2 415.7163} C_DIS
LIN {X 101.6752,Y 66.1595,Z 136,A 28.6791,B 24.9456,C -1.7023,E1 25.1345,E2 417.4552} C_DIS
LIN {X 103.6014,Y 63.1017,Z 136,A 26.9048,B 24.9462,C -1.6944,E1 25.1371,E2 419.2391} C_DIS
LIN {X 105.2458,Y 60.3183,Z 136,A 25.4603,B 24.9462,C -1.6943,E1 25.1392,E2 420.6765} C_DIS
LIN {X 106.6916,Y 57.7231,Z 136,A 23.908,B 24.9469,C -1.6831,E1 25.1413,E2 422.2471} C_DIS
LIN {X 108.3495,Y 54.5449,Z 136,A 22.2364,B 24.9472,C -1.6793,E1 25.1434,E2 423.9185} C_DIS
LIN {X 110.0228,Y 51.0832,Z 136,A 20.5753,B 24.947,C -1.6818,E1 25.1454,E2 425.565} C_DIS
LIN {X 111.3459,Y 48.1307,Z 136,A 18.9892,B 24.9475,C -1.6745,E1 25.1472,E2 427.1597} C_DIS
LIN {X 112.8599,Y 44.4684,Z 136,A 16.9898,B 24.9482,C -1.6626,E1 25.1493,E2 429.176} C_DIS
LIN {X 114.2125,Y 40.8666,Z 136,A 15.3878,B 24.9479,C -1.6678,E1 25.1508,E2 430.7569} C_DIS
LIN {X 115.2354,Y 37.8881,Z 136,A 13.7458,B 24.9486,C -1.6556,E1 25.1523,E2 432.4183} C_DIS
LIN {X 116.506,Y 33.7783,Z 136,A 11.8933,B 24.9485,C -1.6582,E1 25.1537,E2 434.254} C_DIS
LIN {X 117.453,Y 30.3243,Z 136,A 10.0859,B 24.9492,C -1.6472,E1 25.1551,E2 436.077} C_DIS
LIN {X 118.3791,Y 26.4802,Z 136,A 8.2097,B 24.9495,C -1.6409,E1 25.1562,E2 437.9572} C_DIS
LIN {X 119.1486,Y 22.7628,Z 136,A 6.5787,B 24.9495,C -1.6432,E1 25.1571,E2 439.5731} C_DIS
LIN {X 119.7566,Y 19.3217,Z 136,A 4.9283,B 24.9497,C -1.6379,E1 25.1579,E2 441.2264} C_DIS
LIN {X 120.2765,Y 15.7522,Z 136,A 3.1981,B 24.9501,C -1.6312,E1 25.1586,E2 442.9623} C_DIS
LIN {X 120.72,Y 11.8889,Z 136,A 1.2673,B 24.9508,C -1.6205,E1 25.1592,E2 444.9068} C_DIS
LIN {X 121.0751,Y 7.4428,Z 136,A -0.7143,B 24.9508,C -1.6199,E1 25.1595,E2 446.8781} C_DIS
LIN {X 121.251,Y 3.5832,Z 136,A -2.5905,B 24.9513,C -1.6114,E1 25.1597,E2 448.7632} C_DIS
LIN {X 121.3042,Y 0.1958,Z 136,A -4.1006,B 24.9513,C -1.6106,E1 25.1597,E2 450.2662} C_DIS
LIN {X 121.251,Y -3.5832,Z 136,A -5.9973,B 24.9521,C -1.5992,E1 25.1597,E2 452.1785} C_DIS
LIN {X 121.0751,Y -7.443,Z 136,A -7.7446,B 24.9522,C -1.597,E1 25.1594,E2 453.9204} C_DIS
LIN {X 120.72,Y -11.889,Z 136,A -9.8761,B 24.9527,C -1.5889,E1 25.1589,E2 456.0586} C_DIS
LIN {X 120.2814,Y -15.7142,Z 136,A -11.5589,B 24.9527,C -1.5897,E1 25.1583,E2 457.7295} C_DIS
LIN {X 119.8859,Y -18.4909,Z 136,A -12.9097,B 24.953,C -1.584,E1 25.1578,E2 459.0856} C_DIS
LIN {X 119.2516,Y -22.2239,Z 136,A -14.6576,B 24.9532,C -1.5802,E1 25.1569,E2 460.8325} C_DIS
LIN {X 118.5419,Y -25.7367,Z 136,A -16.3654,B 24.9536,C -1.5739,E1 25.1559,E2 462.545} C_DIS
LIN {X 117.6678,Y -29.478,Z 136,A -18.2053,B 24.954,C -1.5668,E1 25.1547,E2 464.3911} C_DIS
LIN {X 116.6753,Y -33.1917,Z 136,A -20.0866,B 24.9545,C -1.5576,E1 25.1533,E2 466.2831} C_DIS
LIN {X 115.5588,Y -36.8874,Z 136,A -21.8434,B 24.9547,C -1.5552,E1 25.1519,E2 468.0358} C_DIS
LIN {X 114.4179,Y -40.2914,Z 136,A -23.4336,B 24.9547,C -1.555,E1 25.1504,E2 469.6175} C_DIS
LIN {X 113.5253,Y -42.738,Z 136,A -24.7046,B 24.955,C -1.5491,E1 25.1492,E2 470.8952} C_DIS
LIN {X 112.2964,Y -45.8728,Z 136,A -26.2377,B 24.9552,C -1.5469,E1 25.1476,E2 472.4249} C_DIS
LIN {X 110.8952,Y -49.162,Z 136,A -28.0539,B 24.9558,C -1.5354,E1 25.1456,E2 474.2585} C_DIS
LIN {X 109.2818,Y -52.6509,Z 136,A -29.7198,B 24.9558,C -1.5372,E1 25.1436,E2 475.911} C_DIS
LIN {X 107.9603,Y -55.3094,Z 136,A -31.1932,B 24.9562,C -1.5295,E1 25.1417,E2 477.3949} C_DIS
LIN {X 105.9093,Y -59.146,Z 136,A -33.298,B 24.9567,C -1.5208,E1 25.1389,E2 479.5091} C_DIS
LIN {X 103.7513,Y -62.8537,Z 136,A -35.218,B 24.9567,C -1.5201,E1 25.1362,E2 481.4208} C_DIS
LIN {X 102.0104,Y -65.6421,Z 136,A -36.7116,B 24.9567,C -1.5186,E1 25.134,E2 482.9106} C_DIS
LIN {X 100.0304,Y -68.621,Z 136,A -38.3885,B 24.957,C -1.5144,E1 25.1314,E2 484.5891} C_DIS
LIN {X 97.9522,Y -71.5568,Z 136,A -40.1701,B 24.9575,C -1.5055,E1 25.1284,E2 486.3829} C_DIS
LIN {X 95.601,Y -74.6691,Z 136,A -42.0048,B 24.9578,C -1.5008,E1 25.1253,E2 488.2199} C_DIS
LIN {X 93.0946,Y -77.7713,Z 136,A -43.9298,B 24.9582,C -1.4938,E1 25.1219,E2 490.1528} C_DIS
LIN {X 90.107,Y -81.2144,Z 136,A -46.0692,B 24.9585,C -1.4888,E1 25.1179,E2 492.2942} C_DIS
LIN {X 87.345,Y -84.1774,Z 136,A -47.975,B 24.9587,C -1.4843,E1 25.1143,E2 494.2023} C_DIS
LIN {X 84.1777,Y -87.3447,Z 136,A -50.0275,B 24.9588,C -1.4822,E1 25.1102,E2 496.2512} C_DIS
LIN {X 81.3963,Y -89.9421,Z 136,A -51.8309,B 24.9591,C -1.4776,E1 25.1065,E2 498.0581} C_DIS
LIN {X 78.2802,Y -92.6675,Z 136,A -53.7248,B 24.9591,C -1.4761,E1 25.1025,E2 499.9482} C_DIS
LIN {X 75.212,Y -95.1745,Z 136,A -55.6864,B 24.9597,C -1.4675,E1 25.0982,E2 501.9227} C_DIS
LIN {X 71.8572,Y -97.7315,Z 136,A -57.5849,B 24.9597,C -1.4678,E1 25.0939,E2 503.8137} C_DIS
LIN {X 68.6667,Y -99.999,Z 136,A -59.3611,B 24.9597,C -1.4675,E1 25.0899,E2 505.5845} C_DIS
LIN {X 65.6438,Y -102.0093,Z 136,A -61.221,B 24.9602,C -1.457,E1 25.0855,E2 507.4629} C_DIS
LIN {X 62.3647,Y -104.0464,Z 136,A -62.9571,B 24.9602,C -1.4578,E1 25.0814,E2 509.1918} C_DIS
LIN {X 58.9943,Y -105.9937,Z 136,A -64.696,B 24.9602,C -1.4593,E1 25.0772,E2 510.9221} C_DIS
LIN {X 55.8515,Y -107.6822,Z 136,A -66.3913,B 24.9602,C -1.4558,E1 25.073,E2 512.6206} C_DIS
LIN {X 53.2007,Y -109.0157,Z 136,A -67.8022,B 24.9604,C -1.4531,E1 25.0695,E2 514.0344} C_DIS
LIN {X 49.722,Y -110.6447,Z 136,A -69.709,B 24.9608,C -1.4458,E1 25.0646,E2 515.9536} C_DIS
LIN {X 46.4149,Y -112.0726,Z 136,A -71.3967,B 24.9609,C -1.4439,E1 25.0602,E2 517.6417} C_DIS
LIN {X 42.8359,Y -113.4886,Z 136,A -73.1792,B 24.9609,C -1.443,E1 25.0556,E2 519.4223} C_DIS
LIN {X 39.4599,Y -114.7061,Z 136,A -74.9006,B 24.9612,C -1.4396,E1 25.0511,E2 521.1485} C_DIS
LIN {X 35.782,Y -115.9062,Z 136,A -76.7371,B 24.9613,C -1.4369,E1 25.0462,E2 522.9879} C_DIS
LIN {X 32.3499,Y -116.9107,Z 136,A -78.4103,B 24.9613,C -1.4358,E1 25.0417,E2 524.6609} C_DIS
LIN {X 28.6313,Y -117.8763,Z 136,A -80.2213,B 24.9615,C -1.4341,E1 25.0368,E2 526.4732} C_DIS
LIN {X 24.5473,Y -118.7944,Z 136,A -82.1505,B 24.9615,C -1.4345,E1 25.0315,E2 528.3989} C_DIS
LIN {X 21.341,Y -119.4115,Z 136,A -83.6492,B 24.9615,C -1.4353,E1 25.0274,E2 529.894} C_DIS
LIN {X 17.7886,Y -119.9938,Z 136,A -85.4872,B 24.9618,C -1.4275,E1 25.0223,E2 531.7486} C_DIS
LIN {X 13.9738,Y -120.4967,Z 136,A -87.238,B 24.9618,C -1.4295,E1 25.0174,E2 533.4934} C_DIS
LIN {X 9.5333,Y -120.9304,Z 136,A -89.2512,B 24.9615,C -1.4328,E1 25.0119,E2 535.4976} C_DIS
LIN {X 6.3941,Y -121.1354,Z 136,A -90.7702,B 24.9617,C -1.4307,E1 25.0076,E2 537.0212} C_DIS
LIN {X 2.968,Y -121.2681,Z 136,A -92.4821,B 24.9619,C -1.4258,E1 25.0028,E2 538.7442} C_DIS
LIN {X 2.968,Y -121.2681,Z 136,A -92.4821,B 24.9619,C -1.4258,E1 25.0028,E2 538.7442} C_DIS
Enddeposition()
LIN {X 0.8999,Y -126.6905,Z 137,A -92.7578,B 24.9647,C -1.373,E1 25.0017,E2 539.145} C_DIS
Startdeposition()
$VEL.CP = VEL_PRINT
LIN {X -1.871,Y -126.6822,Z 137,A -94.418,B 24.9657,C -1.3526,E1 24.9969,E2 540.8536} C_DIS
LIN {X -5.1764,Y -126.5902,Z 137,A -95.8942,B 24.9657,C -1.3533,E1 24.9928,E2 542.3282} C_DIS
LIN {X -8.0266,Y -126.4414,Z 137,A -97.1579,B 24.9657,C -1.3546,E1 24.9893,E2 543.5893} C_DIS
LIN {X -11.5479,Y -126.1695,Z 137,A -98.8953,B 24.966,C -1.3478,E1 24.9844,E2 545.3437} C_DIS
LIN {X -14.9016,Y -125.8162,Z 137,A -100.3415,B 24.9658,C -1.3518,E1 24.9804,E2 546.7811} C_DIS
LIN {X -18.1682,Y -125.3864,Z 137,A -101.7764,B 24.9656,C -1.3549,E1 24.9765,E2 548.21} C_DIS
LIN {X -21.0976,Y -124.9268,Z 137,A -103.1651,B 24.9657,C -1.3529,E1 24.9726,E2 549.6045} C_DIS
LIN {X -24.0843,Y -124.3856,Z 137,A -104.4909,B 24.9656,C -1.3557,E1 24.969,E2 550.9252} C_DIS
LIN {X -26.9849,Y -123.7886,Z 137,A -105.879,B 24.9656,C -1.354,E1 24.9652,E2 552.3191} C_DIS
LIN {X -29.7484,Y -123.1535,Z 137,A -107.1541,B 24.9656,C -1.355,E1 24.9617,E2 553.5935} C_DIS
LIN {X -32.8933,Y -122.3512,Z 137,A -108.6011,B 24.9656,C -1.3569,E1 24.9578,E2 555.038} C_DIS
LIN {X -36.3393,Y -121.3745,Z 137,A -110.2301,B 24.9655,C -1.3575,E1 24.9535,E2 556.6683} C_DIS
LIN {X -38.749,Y -120.6245,Z 137,A -111.3834,B 24.9655,C -1.3579,E1 24.9504,E2 557.8228} C_DIS
LIN {X -41.7238,Y -119.6281,Z 137,A -112.8023,B 24.9655,C -1.3591,E1 24.9466,E2 559.2415} C_DIS
LIN {X -44.6859,Y -118.5535,Z 137,A -114.2808,B 24.9655,C -1.3578,E1 24.9427,E2 560.726} C_DIS
LIN {X -47.6803,Y -117.3814,Z 137,A -115.7276,B 24.9654,C -1.3596,E1 24.939,E2 562.1717} C_DIS
LIN {X -51.8754,Y -115.5883,Z 137,A -117.7737,B 24.9652,C -1.3627,E1 24.9338,E2 564.2153} C_DIS
LIN {X -54.9062,Y -114.1801,Z 137,A -119.3183,B 24.9652,C -1.3629,E1 24.9299,E2 565.7633} C_DIS
LIN {X -57.905,Y -112.6894,Z 137,A -120.9436,B 24.9654,C -1.3596,E1 24.9258,E2 567.4008} C_DIS
LIN {X -61.8425,Y -110.579,Z 137,A -122.9505,B 24.9652,C -1.363,E1 24.9209,E2 569.4054} C_DIS
LIN {X -65.8442,Y -108.2442,Z 137,A -125.023,B 24.965,C -1.3672,E1 24.9159,E2 571.4743} C_DIS
LIN {X -69.388,Y -106.0074,Z 137,A -126.9713,B 24.965,C -1.3677,E1 24.9113,E2 573.4277} C_DIS
LIN {X -73.2114,Y -103.4035,Z 137,A -129.0191,B 24.9647,C -1.3733,E1 24.9066,E2 575.4691} C_DIS
LIN {X -76.6448,Y -100.8855,Z 137,A -130.987,B 24.9647,C -1.3747,E1 24.9022,E2 577.4406} C_DIS
LIN {X -79.8573,Y -98.3622,Z 137,A -132.8591,B 24.9645,C -1.377,E1 24.8981,E2 579.3142} C_DIS
LIN {X -83.2076,Y -95.544,Z 137,A -134.7985,B 24.9642,C -1.3828,E1 24.894,E2 581.2474} C_DIS
LIN {X -86.4443,Y -92.6258,Z 137,A -136.7255,B 24.9639,C -1.3889,E1 24.8901,E2 583.1677} C_DIS
LIN {X -89.1698,Y -90.0051,Z 137,A -138.5116,B 24.9639,C -1.3889,E1 24.8865,E2 584.961} C_DIS
LIN {X -92.0645,Y -87.0418,Z 137,A -140.3836,B 24.9636,C -1.3932,E1 24.8829,E2 586.8311} C_DIS
LIN {X -94.7413,Y -84.1208,Z 137,A -142.217,B 24.9636,C -1.3954,E1 24.8794,E2 588.6675} C_DIS
LIN {X -97.7491,Y -80.606,Z 137,A -144.2789,B 24.9632,C -1.4017,E1 24.8757,E2 590.7238} C_DIS
LIN {X -100.3572,Y -77.335,Z 137,A -146.2211,B 24.9631,C -1.404,E1 24.8724,E2 592.6696} C_DIS
LIN {X -102.8251,Y -74.0223,Z 137,A -148.0915,B 24.9628,C -1.4086,E1 24.8693,E2 594.5382} C_DIS
LIN {X -105.1483,Y -70.6835,Z 137,A -149.8862,B 24.9625,C -1.4154,E1 24.8665,E2 596.3256} C_DIS
LIN {X -107.3563,Y -67.2825,Z 137,A -151.7289,B 24.9622,C -1.4199,E1 24.8637,E2 598.167} C_DIS
LIN {X -109.447,Y -63.8253,Z 137,A -153.5172,B 24.9619,C -1.4266,E1 24.8612,E2 599.9485} C_DIS
LIN {X -111.4185,Y -60.3177,Z 137,A -155.4615,B 24.9619,C -1.4259,E1 24.8585,E2 601.9046} C_DIS
LIN {X -113.0011,Y -57.2927,Z 137,A -156.8843,B 24.9614,C -1.4358,E1 24.8567,E2 603.3114} C_DIS
LIN {X -114.4343,Y -54.374,Z 137,A -158.3636,B 24.9612,C -1.4396,E1 24.8549,E2 604.7897} C_DIS
LIN {X -115.7621,Y -51.4868,Z 137,A -159.8208,B 24.961,C -1.4429,E1 24.8533,E2 606.2472} C_DIS
LIN {X -116.9937,Y -48.623,Z 137,A -161.2217,B 24.9608,C -1.4474,E1 24.8517,E2 607.645} C_DIS
LIN {X -118.1821,Y -45.6591,Z 137,A -162.7201,B 24.9607,C -1.4493,E1 24.8502,E2 609.1474} C_DIS
LIN {X -119.3016,Y -42.649,Z 137,A -164.122,B 24.9603,C -1.4559,E1 24.8489,E2 610.5414} C_DIS
LIN {X -120.4513,Y -39.2911,Z 137,A -165.7406,B 24.9601,C -1.4602,E1 24.8474,E2 612.1591} C_DIS
Enddeposition()
END
